KUKA KRL program: EPS_2_25362_MH3A_A_20251103083056.src

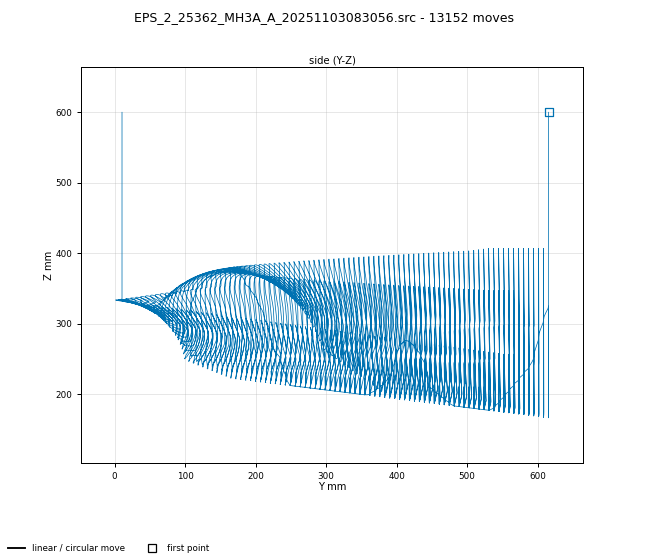
[picture p0: tool path of EPS_2_25362_MH3A_A_20251103083056.src, 13152 of 13154 moves have a stored position in this frame; points joined in program order, loops and branches not executed]
&ACCESS RVP
&REL 4
&COMMENT QRS 19112012
&PARAM EDITMASK = *
DEF PART()
EXT BAS (BAS_COMMAND :IN,REAL :IN )
INT I
BAS (#INITMOV,0 )

;KUKA QRS Post kuka4.cps  Date:22-06-2017 !

File_ID=2900

QRS_PRE_INIT()

;Init var - Until changes are made in qrs_pre_init
Outlet_Square_prg=0
Inlet_1_Square_prg=0
Inlet_2_Square_prg=0
Inlet_3_Square_prg=0
Inlet_4_Square_prg=0
Inlet_5_Square_prg=0

Outlet_1={X 0.000, Y 531.880, Z 306.500, B 0.000, E1 0.000 }
Inlet_1={X 0.000, Y 536.220, Z 246.500, B 0.000, E1 90.000 }
Inlet_2={X 0.000, Y 550.320, Z 206.500, B 0.000, E1 180.000 }
Outlet_1_type=201
Inlet_1_type=201
Inlet_2_type=101
;QRS#1=Sidecore dimensions
;QRS#2=200-8" PVC SDR 35
;QRS#3=200-8" PVC SDR 35
;QRS#4=100-4" PVC SDR 28
;QRS#5=
;QRS#6=
;QRS#7=
;QRS#8=
;QRS#9=12-08 PSX
;QRS#10=12-08 PSX
;QRS#11=8QRS PSX
;QRS#12=
;QRS#13=
;QRS#14=
;QRS#15=
;QRS#16=1220x127x686 2,25'
;QRS#17=EPS Height
;QRS#18=407
;QRS#19=*
;QRS#20= UPDATED VERSION 22-06-2017
;QRS#21=*
Outlet_Square=0100
Inlet_1_Square=0100
Inlet_2_Square=045
Inlet_3_Square=0
Inlet_4_Square=0
Inlet_5_Square=0
Mill_Square=1
Outlet_Square_Prg=204
Inlet_1_Square_prg=204
Inlet_2_Square_prg=201

QRS_INIT()

$ADVANCE=5

; T1
PTP {E1 173.498,E2 173.498}
PTP {X 0,Y 615.498,A -85,B 0,C 180,E1 173.498,E2 173.498,E3 0,E4 0,E5 0,E6 0}
QRS_SPEED_INIT()
LIN {X 0,Y 615.498,Z 600,A -85,B 0,C 180,E1 173.498,E2 173.498,E3 0,E4 0,E5 0,E6 0} C_VEL
LIN {X 0,Y 615.498,Z 337.732,A -85,B 0,C 180,E1 173.498,E2 173.498} C_VEL
LIN {X 0,Y 615.498,Z 326.853,A -85,B 0,C 180,E1 173.498,E2 173.498} C_VEL
LIN {X 0,Y 615.496,Z 325.209,A -85,B 0,C 180,E1 173.418,E2 173.418} C_VEL
LIN {X 0,Y 615.497,Z 317.536,A -85,B 0,C 180,E1 172.455,E2 172.455} C_VEL
LIN {X 0,Y 615.498,Z 307.758,A -85,B 0,C 180,E1 171.463,E2 171.463} C_VEL
LIN {X 0,Y 615.498,Z 297.492,A -85,B 0,C 180,E1 170.636,E2 170.636} C_VEL
LIN {X 0,Y 615.449,Z 285.935,A -85,B 0,C 180,E1 169.888,E2 169.888} C_VEL
LIN {X 0,Y 615.45,Z 274.237,A -85,B 0,C 180,E1 169.299,E2 169.299} C_VEL
LIN {X 0,Y 615.495,Z 262.393,A -85,B 0,C 180,E1 168.847,E2 168.847} C_VEL
LIN {X 0,Y 615.488,Z 250.38,A -85,B 0,C 180,E1 168.515,E2 168.515} C_VEL
LIN {X 0,Y 615.473,Z 240.081,A -85,B 0,C 180,E1 168.306,E2 168.306} C_VEL
LIN {X 0,Y 615.432,Z 231.733,A -85,B 0,C 180,E1 165.768,E2 165.768} C_VEL
LIN {X 0,Y 615.485,Z 222.926,A -85,B 0,C 180,E1 163.072,E2 163.072} C_VEL
LIN {X 0,Y 615.428,Z 214.085,A -85,B 0,C 180,E1 160.313,E2 160.313} C_VEL
LIN {X 0,Y 615.422,Z 206.32,A -85,B 0,C 180,E1 157.861,E2 157.861} C_VEL
LIN {X 0,Y 615.473,Z 197.446,A -85,B 0,C 180,E1 155.007,E2 155.007} C_VEL
LIN {X 0,Y 615.429,Z 189.685,A -85,B 0,C 180,E1 152.451,E2 152.451} C_VEL
LIN {X 0,Y 615.495,Z 181.752,A -85,B 0,C 180,E1 149.84,E2 149.84} C_VEL
LIN {X 0,Y 615.493,Z 173.403,A -85,B 0,C 180,E1 147.154,E2 147.154} C_VEL
LIN {X 0,Y 615.459,Z 166.7,A -85,B 0,C 180,E1 144.983,E2 144.983} C_VEL
LIN {X 0,Y 615.455,Z 166.697,A -85,B 0,C 180,E1 142.755,E2 142.755} C_VEL
LIN {X 0,Y 615.482,Z 166.691,A -85,B 0,C 180,E1 139.912,E2 139.912} C_VEL
LIN {X 0,Y 615.499,Z 166.691,A -85,B 0,C 180,E1 137.648,E2 137.648} C_VEL
LIN {X 0,Y 615.44,Z 166.7,A -85,B 0,C 180,E1 134.927,E2 134.927} C_VEL
LIN {X 0,Y 615.493,Z 166.697,A -85,B 0,C 180,E1 132.353,E2 132.353} C_VEL
LIN {X 0,Y 615.492,Z 166.691,A -85,B 0,C 180,E1 129.75,E2 129.75} C_VEL
LIN {X 0,Y 615.44,Z 166.7,A -85,B 0,C 180,E1 126.93,E2 126.93} C_VEL
LIN {X 0,Y 615.468,Z 166.701,A -85,B 0,C 180,E1 124.697,E2 124.697} C_VEL
LIN {X 0,Y 615.489,Z 166.691,A -85,B 0,C 180,E1 122.33,E2 122.33} C_VEL
LIN {X 0,Y 615.494,Z 166.701,A -85,B 0,C 180,E1 119.795,E2 119.795} C_VEL
LIN {X 0,Y 615.491,Z 170.653,A -85,B 0,C 180,E1 117.045,E2 117.045} C_VEL
LIN {X 0,Y 615.49,Z 174.728,A -85,B 0,C 180,E1 114.273,E2 114.273} C_VEL
LIN {X 0,Y 615.467,Z 179.104,A -85,B 0,C 180,E1 111.433,E2 111.433} C_VEL
LIN {X 0,Y 615.482,Z 183.48,A -85,B 0,C 180,E1 108.647,E2 108.647} C_VEL
LIN {X 0,Y 615.48,Z 187.851,A -85,B 0,C 180,E1 105.906,E2 105.906} C_VEL
LIN {X 0,Y 615.448,Z 192.229,A -85,B 0,C 180,E1 103.203,E2 103.203} C_VEL
LIN {X 0,Y 615.496,Z 196.599,A -85,B 0,C 180,E1 100.528,E2 100.528} C_VEL
LIN {X 0,Y 615.436,Z 200.972,A -85,B 0,C 180,E1 97.877,E2 97.877} C_VEL
LIN {X 0,Y 615.491,Z 202.929,A -85,B 0,C 180,E1 96.693,E2 96.693} C_VEL
LIN {X 0,Y 615.467,Z 211.517,A -85,B 0,C 180,E1 96.393,E2 96.393} C_VEL
LIN {X 0,Y 615.433,Z 219.944,A -85,B 0,C 180,E1 95.982,E2 95.982} C_VEL
LIN {X 0,Y 615.434,Z 227.673,A -85,B 0,C 180,E1 95.489,E2 95.489} C_VEL
LIN {X 0,Y 615.485,Z 234.509,A -85,B 0,C 180,E1 94.914,E2 94.914} C_VEL
LIN {X 0,Y 615.497,Z 240.661,A -85,B 0,C 180,E1 94.257,E2 94.257} C_VEL
LIN {X 0,Y 615.497,Z 245.51,A -85,B 0,C 180,E1 93.601,E2 93.601} C_VEL
LIN {X 0,Y 615.498,Z 249.246,A -85,B 0,C 180,E1 92.946,E2 92.946} C_VEL
LIN {X 0,Y 615.498,Z 253.227,A -85,B 0,C 180,E1 91.964,E2 91.964} C_VEL
LIN {X 0,Y 615.496,Z 254.962,A -85,B 0,C 180,E1 91.309,E2 91.309} C_VEL
LIN {X 0,Y 615.496,Z 256.003,A -85,B 0,C 180,E1 90.655,E2 90.655} C_VEL
LIN {X 0,Y 615.494,Z 256.384,A -85,B 0,C 180,E1 90.001,E2 90.001} C_VEL
LIN {X 0,Y 615.496,Z 256.106,A -85,B 0,C 180,E1 89.347,E2 89.347} C_VEL
LIN {X 0,Y 615.497,Z 255.167,A -85,B 0,C 180,E1 88.692,E2 88.692} C_VEL
LIN {X 0,Y 615.496,Z 253.539,A -85,B 0,C 180,E1 88.038,E2 88.038} C_VEL
LIN {X 0,Y 615.497,Z 251.17,A -85,B 0,C 180,E1 87.383,E2 87.383} C_VEL
LIN {X 0,Y 615.498,Z 246.077,A -85,B 0,C 180,E1 86.4,E2 86.4} C_VEL
LIN {X 0,Y 615.498,Z 240.038,A -85,B 0,C 180,E1 85.58,E2 85.58} C_VEL
LIN {X 0,Y 615.468,Z 233.768,A -85,B 0,C 180,E1 84.924,E2 84.924} C_VEL
LIN {X 0,Y 615.422,Z 226.618,A -85,B 0,C 180,E1 84.348,E2 84.348} C_VEL
LIN {X 0,Y 615.432,Z 218.637,A -85,B 0,C 180,E1 83.855,E2 83.855} C_VEL
LIN {X 0,Y 615.473,Z 209.487,A -85,B 0,C 180,E1 83.437,E2 83.437} C_VEL
LIN {X 0,Y 615.499,Z 202.92,A -85,B 0,C 180,E1 83.213,E2 83.213} C_VEL
LIN {X 0,Y 615.447,Z 198.945,A -85,B 0,C 180,E1 80.802,E2 80.802} C_VEL
LIN {X 0,Y 615.446,Z 195.663,A -85,B 0,C 180,E1 78.807,E2 78.807} C_VEL
LIN {X 0,Y 615.443,Z 192.381,A -85,B 0,C 180,E1 76.799,E2 76.799} C_VEL
LIN {X 0,Y 615.445,Z 189.098,A -85,B 0,C 180,E1 74.774,E2 74.774} C_VEL
LIN {X 0,Y 615.484,Z 184.718,A -85,B 0,C 180,E1 72.044,E2 72.044} C_VEL
LIN {X 0,Y 615.47,Z 180.343,A -85,B 0,C 180,E1 69.27,E2 69.27} C_VEL
LIN {X 0,Y 615.48,Z 175.962,A -85,B 0,C 180,E1 66.445,E2 66.445} C_VEL
LIN {X 0,Y 615.493,Z 171.632,A -85,B 0,C 180,E1 63.557,E2 63.557} C_VEL
LIN {X 0,Y 615.493,Z 168.479,A -85,B 0,C 180,E1 61.344,E2 61.344} C_VEL
LIN {X 0,Y 615.497,Z 166.83,A -85,B 0,C 180,E1 60.204,E2 60.204} C_VEL
LIN {X 0,Y 615.464,Z 166.689,A -85,B 0,C 180,E1 57.543,E2 57.543} C_VEL
LIN {X 0,Y 615.454,Z 166.693,A -85,B 0,C 180,E1 55.184,E2 55.184} C_VEL
LIN {X 0,Y 615.479,Z 166.7,A -85,B 0,C 180,E1 52.759,E2 52.759} C_VEL
LIN {X 0,Y 615.48,Z 166.686,A -85,B 0,C 180,E1 49.912,E2 49.912} C_VEL
LIN {X 0,Y 615.463,Z 166.69,A -85,B 0,C 180,E1 47.647,E2 47.647} C_VEL
LIN {X 0,Y 615.498,Z 166.699,A -85,B 0,C 180,E1 44.934,E2 44.934} C_VEL
LIN {X 0,Y 615.475,Z 166.686,A -85,B 0,C 180,E1 42.081,E2 42.081} C_VEL
LIN {X 0,Y 615.47,Z 166.692,A -85,B 0,C 180,E1 39.752,E2 39.752} C_VEL
LIN {X 0,Y 615.484,Z 166.691,A -85,B 0,C 180,E1 36.938,E2 36.938} C_VEL
LIN {X 0,Y 615.489,Z 166.684,A -85,B 0,C 180,E1 34.703,E2 34.703} C_VEL
LIN {X 0,Y 615.481,Z 166.686,A -85,B 0,C 180,E1 32.332,E2 32.332} C_VEL
LIN {X 0,Y 615.489,Z 166.698,A -85,B 0,C 180,E1 29.797,E2 29.797} C_VEL
LIN {X 0,Y 615.477,Z 166.687,A -85,B 0,C 180,E1 27.046,E2 27.046} C_VEL
LIN {X 0,Y 615.483,Z 166.693,A -85,B 0,C 180,E1 24.272,E2 24.272} C_VEL
LIN {X 0,Y 615.472,Z 166.69,A -85,B 0,C 180,E1 21.433,E2 21.433} C_VEL
LIN {X 0,Y 615.486,Z 166.69,A -85,B 0,C 180,E1 18.608,E2 18.608} C_VEL
LIN {X 0,Y 615.471,Z 166.694,A -85,B 0,C 180,E1 15.906,E2 15.906} C_VEL
LIN {X 0,Y 615.49,Z 166.684,A -85,B 0,C 180,E1 13.201,E2 13.201} C_VEL
LIN {X 0,Y 615.489,Z 166.702,A -85,B 0,C 180,E1 10.527,E2 10.527} C_VEL
LIN {X 0,Y 615.459,Z 166.691,A -85,B 0,C 180,E1 7.876,E2 7.876} C_VEL
LIN {X 0,Y 615.496,Z 166.688,A -85,B 0,C 180,E1 5.241,E2 5.241} C_VEL
LIN {X 0,Y 615.47,Z 166.697,A -85,B 0,C 180,E1 2.618,E2 2.618} C_VEL
LIN {X 0,Y 615.456,Z 166.691,A -85,B 0,C 180,E1 0,E2 0} C_VEL
LIN {X 0,Y 615.495,Z 166.693,A -85,B 0,C 180,E1 -2.618,E2 -2.618} C_VEL
LIN {X 0,Y 615.451,Z 166.697,A -85,B 0,C 180,E1 -5.242,E2 -5.242} C_VEL
LIN {X 0,Y 615.446,Z 166.696,A -85,B 0,C 180,E1 -7.216,E2 -7.216} C_VEL
LIN {X 0,Y 615.442,Z 166.696,A -85,B 0,C 180,E1 -9.199,E2 -9.199} C_VEL
LIN {X 0,Y 615.437,Z 166.696,A -85,B 0,C 180,E1 -11.194,E2 -11.194} C_VEL
LIN {X 0,Y 615.473,Z 166.694,A -85,B 0,C 180,E1 -13.933,E2 -13.933} C_VEL
LIN {X 0,Y 615.453,Z 166.699,A -85,B 0,C 180,E1 -16.588,E2 -16.588} C_VEL
LIN {X 0,Y 615.439,Z 166.699,A -85,B 0,C 180,E1 -18.648,E2 -18.648} C_VEL
LIN {X 0,Y 615.427,Z 166.699,A -85,B 0,C 180,E1 -20.733,E2 -20.733} C_VEL
LIN {X 0,Y 615.419,Z 166.699,A -85,B 0,C 180,E1 -22.847,E2 -22.847} C_VEL
LIN {X 0,Y 615.418,Z 166.7,A -85,B 0,C 180,E1 -24.995,E2 -24.995} C_VEL
LIN {X 0,Y 615.433,Z 166.7,A -85,B 0,C 180,E1 -27.18,E2 -27.18} C_VEL
LIN {X 0,Y 615.438,Z 166.698,A -85,B 0,C 180,E1 -30.163,E2 -30.163} C_VEL
LIN {X 0,Y 615.424,Z 166.698,A -85,B 0,C 180,E1 -32.461,E2 -32.461} C_VEL
LIN {X 0,Y 615.438,Z 166.699,A -85,B 0,C 180,E1 -34.818,E2 -34.818} C_VEL
LIN {X 0,Y 615.488,Z 166.702,A -85,B 0,C 180,E1 -37.242,E2 -37.242} C_VEL
LIN {X 0,Y 615.457,Z 166.694,A -85,B 0,C 180,E1 -39.753,E2 -39.753} C_VEL
LIN {X 0,Y 615.44,Z 166.696,A -85,B 0,C 180,E1 -42.357,E2 -42.357} C_VEL
LIN {X 0,Y 615.491,Z 166.696,A -85,B 0,C 180,E1 -45.068,E2 -45.068} C_VEL
LIN {X 0,Y 615.454,Z 166.692,A -85,B 0,C 180,E1 -47.646,E2 -47.646} C_VEL
LIN {X 0,Y 615.456,Z 166.697,A -85,B 0,C 180,E1 -50.249,E2 -50.249} C_VEL
LIN {X 0,Y 615.487,Z 166.688,A -85,B 0,C 180,E1 -53.064,E2 -53.064} C_VEL
LIN {X 0,Y 615.467,Z 166.689,A -85,B 0,C 180,E1 -55.303,E2 -55.303} C_VEL
LIN {X 0,Y 615.456,Z 166.693,A -85,B 0,C 180,E1 -57.674,E2 -57.674} C_VEL
LIN {X 0,Y 615.497,Z 166.7,A -85,B 0,C 180,E1 -60.204,E2 -60.204} C_VEL
LIN {X 0,Y 615.46,Z 166.871,A -85,B 0,C 180,E1 -61.448,E2 -61.448} C_VEL
LIN {X 0,Y 615.473,Z 186.055,A -85,B 0,C 180,E1 -64.103,E2 -64.103} C_VEL
LIN {X 0,Y 615.484,Z 205.999,A -85,B 0,C 180,E1 -66.801,E2 -66.801} C_VEL
LIN {X 0,Y 615.469,Z 225.967,A -85,B 0,C 180,E1 -69.448,E2 -69.448} C_VEL
LIN {X 0,Y 615.482,Z 247.188,A -85,B 0,C 180,E1 -72.216,E2 -72.216} C_VEL
LIN {X 0,Y 615.481,Z 268.409,A -85,B 0,C 180,E1 -74.944,E2 -74.944} C_VEL
LIN {X 0,Y 615.47,Z 289.61,A -85,B 0,C 180,E1 -77.638,E2 -77.638} C_VEL
LIN {X 0,Y 615.498,Z 294.736,A -85,B 0,C 180,E1 -78.287,E2 -78.287} C_VEL
LIN {X 0,Y 615.483,Z 310.284,A -85,B 0,C 180,E1 -78.558,E2 -78.558} C_VEL
LIN {X 0,Y 615.479,Z 323.353,A -85,B 0,C 180,E1 -78.922,E2 -78.922} C_VEL
LIN {X 0,Y 615.487,Z 335.144,A -85,B 0,C 180,E1 -79.384,E2 -79.384} C_VEL
LIN {X 0,Y 615.481,Z 346.592,A -85,B 0,C 180,E1 -79.973,E2 -79.973} C_VEL
LIN {X 0,Y 615.499,Z 358.034,A -85,B 0,C 180,E1 -80.719,E2 -80.719} C_VEL
LIN {X 0,Y 615.498,Z 367.268,A -85,B 0,C 180,E1 -81.464,E2 -81.464} C_VEL
LIN {X 0,Y 615.5,Z 375.662,A -85,B 0,C 180,E1 -82.291,E2 -82.291} C_VEL
LIN {X 0,Y 615.497,Z 383.692,A -85,B 0,C 180,E1 -83.259,E2 -83.259} C_VEL
LIN {X 0,Y 615.499,Z 389.428,A -85,B 0,C 180,E1 -84.102,E2 -84.102} C_VEL
LIN {X 0,Y 615.496,Z 394.877,A -85,B 0,C 180,E1 -85.088,E2 -85.088} C_VEL
LIN {X 0,Y 615.497,Z 399.144,A -85,B 0,C 180,E1 -86.072,E2 -86.072} C_VEL
LIN {X 0,Y 615.494,Z 401.401,A -85,B 0,C 180,E1 -86.728,E2 -86.728} C_VEL
LIN {X 0,Y 615.497,Z 403.235,A -85,B 0,C 180,E1 -87.383,E2 -87.383} C_VEL
LIN {X 0,Y 615.5,Z 404.609,A -85,B 0,C 180,E1 -88.038,E2 -88.038} C_VEL
LIN {X 0,Y 615.496,Z 406.174,A -85,B 0,C 180,E1 -89.347,E2 -89.347} C_VEL
LIN {X 0,Y 615.494,Z 406.389,A -85,B 0,C 180,E1 -90.001,E2 -90.001} C_VEL
LIN {X 0,Y 615.495,Z 405.579,A -85,B 0,C 180,E1 -91.309,E2 -91.309} C_VEL
LIN {X 0,Y 615.5,Z 404.606,A -85,B 0,C 180,E1 -91.964,E2 -91.964} C_VEL
LIN {X 0,Y 615.497,Z 403.231,A -85,B 0,C 180,E1 -92.619,E2 -92.619} C_VEL
LIN {X 0,Y 615.496,Z 400.347,A -85,B 0,C 180,E1 -93.601,E2 -93.601} C_VEL
LIN {X 0,Y 615.498,Z 396.438,A -85,B 0,C 180,E1 -94.585,E2 -94.585} C_VEL
LIN {X 0,Y 615.499,Z 391.4,A -85,B 0,C 180,E1 -95.57,E2 -95.57} C_VEL
LIN {X 0,Y 615.497,Z 384.87,A -85,B 0,C 180,E1 -96.583,E2 -96.583} C_VEL
LIN {X 0,Y 615.497,Z 377.126,A -85,B 0,C 180,E1 -97.546,E2 -97.546} C_VEL
LIN {X 0,Y 615.498,Z 369.037,A -85,B 0,C 180,E1 -98.372,E2 -98.372} C_VEL
LIN {X 0,Y 615.499,Z 359.157,A -85,B 0,C 180,E1 -99.199,E2 -99.199} C_VEL
LIN {X 0,Y 615.485,Z 347.969,A -85,B 0,C 180,E1 -99.946,E2 -99.946} C_VEL
LIN {X 0,Y 615.485,Z 337.007,A -85,B 0,C 180,E1 -100.528,E2 -100.528} C_VEL
LIN {X 0,Y 615.479,Z 324.491,A -85,B 0,C 180,E1 -101.04,E2 -101.04} C_VEL
LIN {X 0,Y 615.481,Z 312.033,A -85,B 0,C 180,E1 -101.402,E2 -101.402} C_VEL
LIN {X 0,Y 615.497,Z 298.409,A -85,B 0,C 180,E1 -101.653,E2 -101.653} C_VEL
LIN {X 0,Y 615.498,Z 294.722,A -85,B 0,C 180,E1 -101.715,E2 -101.715} C_VEL
LIN {X 0,Y 615.472,Z 272.374,A -85,B 0,C 180,E1 -104.55,E2 -104.55} C_VEL
LIN {X 0,Y 615.481,Z 251.154,A -85,B 0,C 180,E1 -107.271,E2 -107.271} C_VEL
LIN {X 0,Y 615.481,Z 229.912,A -85,B 0,C 180,E1 -110.034,E2 -110.034} C_VEL
LIN {X 0,Y 615.471,Z 210.527,A -85,B 0,C 180,E1 -112.595,E2 -112.595} C_VEL
LIN {X 0,Y 615.498,Z 189.5,A -85,B 0,C 180,E1 -115.425,E2 -115.425} C_VEL
LIN {X 0,Y 615.471,Z 169.523,A -85,B 0,C 180,E1 -118.18,E2 -118.18} C_VEL
LIN {X 0,Y 615.46,Z 166.693,A -85,B 0,C 180,E1 -118.606,E2 -118.606} C_VEL
LIN {X 0,Y 615.484,Z 166.694,A -85,B 0,C 180,E1 -121.085,E2 -121.085} C_VEL
LIN {X 0,Y 615.427,Z 166.7,A -85,B 0,C 180,E1 -124.026,E2 -124.026} C_VEL
LIN {X 0,Y 615.488,Z 166.696,A -85,B 0,C 180,E1 -126.936,E2 -126.936} C_VEL
LIN {X 0,Y 615.459,Z 166.695,A -85,B 0,C 180,E1 -129.753,E2 -129.753} C_VEL
LIN {X 0,Y 615.488,Z 166.694,A -85,B 0,C 180,E1 -132.354,E2 -132.354} C_VEL
LIN {X 0,Y 615.484,Z 166.69,A -85,B 0,C 180,E1 -135.069,E2 -135.069} C_VEL
LIN {X 0,Y 615.476,Z 166.697,A -85,B 0,C 180,E1 -137.646,E2 -137.646} C_VEL
LIN {X 0,Y 615.465,Z 166.692,A -85,B 0,C 180,E1 -140.248,E2 -140.248} C_VEL
LIN {X 0,Y 615.452,Z 166.7,A -85,B 0,C 180,E1 -143.068,E2 -143.068} C_VEL
LIN {X 0,Y 615.433,Z 166.7,A -85,B 0,C 180,E1 -145.642,E2 -145.642} C_VEL
LIN {X 0,Y 615.449,Z 166.873,A -85,B 0,C 180,E1 -145.893,E2 -145.893} C_VEL
LIN {X 0,Y 615.494,Z 175.891,A -85,B 0,C 180,E1 -148.315,E2 -148.315} C_VEL
LIN {X 0,Y 615.464,Z 184.98,A -85,B 0,C 180,E1 -150.967,E2 -150.967} C_VEL
LIN {X 0,Y 615.489,Z 192.732,A -85,B 0,C 180,E1 -153.556,E2 -153.556} C_VEL
LIN {X 0,Y 615.479,Z 201.605,A -85,B 0,C 180,E1 -156.443,E2 -156.443} C_VEL
LIN {X 0,Y 615.491,Z 210.458,A -85,B 0,C 180,E1 -159.269,E2 -159.269} C_VEL
LIN {X 0,Y 615.492,Z 219.321,A -85,B 0,C 180,E1 -162.043,E2 -162.043} C_VEL
LIN {X 0,Y 615.49,Z 228.167,A -85,B 0,C 180,E1 -164.774,E2 -164.774} C_VEL
LIN {X 0,Y 615.474,Z 237.019,A -85,B 0,C 180,E1 -167.47,E2 -167.47} C_VEL
LIN {X 0,Y 615.487,Z 240.126,A -85,B 0,C 180,E1 -168.411,E2 -168.411} C_VEL
LIN {X 0,Y 615.492,Z 253.696,A -85,B 0,C 180,E1 -168.682,E2 -168.682} C_VEL
LIN {X 0,Y 615.468,Z 266.631,A -85,B 0,C 180,E1 -169.084,E2 -169.084} C_VEL
LIN {X 0,Y 615.479,Z 277.823,A -85,B 0,C 180,E1 -169.556,E2 -169.556} C_VEL
LIN {X 0,Y 615.489,Z 290.02,A -85,B 0,C 180,E1 -170.221,E2 -170.221} C_VEL
LIN {X 0,Y 615.498,Z 300.713,A -85,B 0,C 180,E1 -170.967,E2 -170.967} C_VEL
LIN {X 0,Y 615.498,Z 310.33,A -85,B 0,C 180,E1 -171.794,E2 -171.794} C_VEL
LIN {X 0,Y 615.497,Z 318.209,A -85,B 0,C 180,E1 -172.62,E2 -172.62} C_VEL
LIN {X 0,Y 615.497,Z 325.899,A -85,B 0,C 180,E1 -173.608,E2 -173.608} C_VEL
LIN {X 0,Y 615.497,Z 332.958,A -85,B 0,C 180,E1 -174.759,E2 -174.759} C_VEL
LIN {X 0,Y 615.498,Z 337.657,A -85,B 0,C 180,E1 -175.744,E2 -175.744} C_VEL
LIN {X 0,Y 615.494,Z 341.255,A -85,B 0,C 180,E1 -176.727,E2 -176.727} C_VEL
LIN {X 0,Y 615.496,Z 343.115,A -85,B 0,C 180,E1 -177.382,E2 -177.382} C_VEL
LIN {X 0,Y 615.497,Z 344.533,A -85,B 0,C 180,E1 -178.037,E2 -178.037} C_VEL
LIN {X 0,Y 615.497,Z 346.141,A -85,B 0,C 180,E1 -179.346,E2 -179.346} C_VEL
LIN {X 0,Y 615.494,Z 346.384,A -85,B 0,C 180,E1 -180,E2 -180} C_VEL
LIN {X 0,Y 615.495,Z 346.206,A -85,B 0,C 180,E1 -180.654,E2 -180.654} C_VEL
LIN {X 0,Y 615.496,Z 344.683,A -85,B 0,C 180,E1 -181.963,E2 -181.963} C_VEL
LIN {X 0,Y 615.498,Z 343.341,A -85,B 0,C 180,E1 -182.618,E2 -182.618} C_VEL
LIN {X 0,Y 615.497,Z 340.494,A -85,B 0,C 180,E1 -183.601,E2 -183.601} C_VEL
LIN {X 0,Y 615.498,Z 336.634,A -85,B 0,C 180,E1 -184.585,E2 -184.585} C_VEL
LIN {X 0,Y 615.498,Z 331.651,A -85,B 0,C 180,E1 -185.57,E2 -185.57} C_VEL
LIN {X 0,Y 615.496,Z 325.209,A -85,B 0,C 180,E1 -186.582,E2 -186.582} C_VEL
LIN {X 0,Y 614.829,Z 322.027,A -85,B 0,C 180,E1 -187.031,E2 -187.031} C_VEL
LIN {X 0,Y 611.989,Z 316.454,A -85,B 0,C 180,E1 -187.748,E2 -187.748} C_VEL
LIN {X 0,Y 609.138,Z 310.179,A -85,B 0,C 180,E1 -188.429,E2 -188.429} C_VEL
LIN {X 0,Y 608.477,Z 305.938,A -85,B 0,C 180,E1 -188.819,E2 -188.819} C_VEL
LIN {X 0,Y 608.49,Z 295.389,A -85,B 0,C 180,E1 -189.641,E2 -189.641} C_VEL
LIN {X 0,Y 608.446,Z 284.609,A -85,B 0,C 180,E1 -190.314,E2 -190.314} C_VEL
LIN {X 0,Y 608.493,Z 272.214,A -85,B 0,C 180,E1 -190.917,E2 -190.917} C_VEL
LIN {X 0,Y 608.556,Z 259.968,A -85,B 0,C 180,E1 -191.365,E2 -191.365} C_VEL
LIN {X 0,Y 608.538,Z 247.651,A -85,B 0,C 180,E1 -191.681,E2 -191.681} C_VEL
LIN {X 0,Y 608.425,Z 240.5,A -85,B 0,C 180,E1 -191.81,E2 -191.81} C_VEL
LIN {X 0,Y 608.384,Z 232.081,A -85,B 0,C 180,E1 -194.381,E2 -194.381} C_VEL
LIN {X 0,Y 608.444,Z 223.175,A -85,B 0,C 180,E1 -197.13,E2 -197.13} C_VEL
LIN {X 0,Y 608.394,Z 214.268,A -85,B 0,C 180,E1 -199.924,E2 -199.924} C_VEL
LIN {X 0,Y 608.433,Z 206.281,A -85,B 0,C 180,E1 -202.469,E2 -202.469} C_VEL
LIN {X 0,Y 608.417,Z 197.567,A -85,B 0,C 180,E1 -205.303,E2 -205.303} C_VEL
LIN {X 0,Y 608.417,Z 189.772,A -85,B 0,C 180,E1 -207.894,E2 -207.894} C_VEL
LIN {X 0,Y 608.488,Z 181.66,A -85,B 0,C 180,E1 -210.544,E2 -210.544} C_VEL
LIN {X 0,Y 608.475,Z 173.202,A -85,B 0,C 180,E1 -213.274,E2 -213.274} C_VEL
LIN {X 0,Y 608.433,Z 167.696,A -85,B 0,C 180,E1 -215.062,E2 -215.062} C_VEL
LIN {X 0,Y 608.463,Z 167.695,A -85,B 0,C 180,E1 -217.747,E2 -217.747} C_VEL
LIN {X 0,Y 608.451,Z 167.691,A -85,B 0,C 180,E1 -220.328,E2 -220.328} C_VEL
LIN {X 0,Y 608.432,Z 167.697,A -85,B 0,C 180,E1 -222.962,E2 -222.962} C_VEL
LIN {X 0,Y 608.456,Z 167.695,A -85,B 0,C 180,E1 -225.736,E2 -225.736} C_VEL
LIN {X 0,Y 608.459,Z 167.692,A -85,B 0,C 180,E1 -228.658,E2 -228.658} C_VEL
LIN {X 0,Y 608.461,Z 167.691,A -85,B 0,C 180,E1 -231.761,E2 -231.761} C_VEL
LIN {X 0,Y 608.419,Z 167.695,A -85,B 0,C 180,E1 -234.72,E2 -234.72} C_VEL
LIN {X 0,Y 608.463,Z 167.692,A -85,B 0,C 180,E1 -237.478,E2 -237.478} C_VEL
LIN {X 0,Y 608.478,Z 167.693,A -85,B 0,C 180,E1 -240.22,E2 -240.22} C_VEL
LIN {X 0,Y 608.433,Z 171.873,A -85,B 0,C 180,E1 -243.224,E2 -243.224} C_VEL
LIN {X 0,Y 608.43,Z 175.706,A -85,B 0,C 180,E1 -245.858,E2 -245.858} C_VEL
LIN {X 0,Y 608.404,Z 179.457,A -85,B 0,C 180,E1 -248.305,E2 -248.305} C_VEL
LIN {X 0,Y 608.399,Z 182.761,A -85,B 0,C 180,E1 -250.427,E2 -250.427} C_VEL
LIN {X 0,Y 608.394,Z 186.065,A -85,B 0,C 180,E1 -252.521,E2 -252.521} C_VEL
LIN {X 0,Y 608.408,Z 190.471,A -85,B 0,C 180,E1 -255.277,E2 -255.277} C_VEL
LIN {X 0,Y 608.411,Z 194.877,A -85,B 0,C 180,E1 -257.998,E2 -257.998} C_VEL
LIN {X 0,Y 608.392,Z 198.181,A -85,B 0,C 180,E1 -260.021,E2 -260.021} C_VEL
LIN {X 0,Y 608.384,Z 202.587,A -85,B 0,C 180,E1 -262.699,E2 -262.699} C_VEL
LIN {X 0,Y 608.442,Z 203.457,A -85,B 0,C 180,E1 -263.226,E2 -263.226} C_VEL
LIN {X 0,Y 608.431,Z 212.066,A -85,B 0,C 180,E1 -263.533,E2 -263.533} C_VEL
LIN {X 0,Y 608.391,Z 220.456,A -85,B 0,C 180,E1 -263.948,E2 -263.948} C_VEL
LIN {X 0,Y 608.403,Z 228.169,A -85,B 0,C 180,E1 -264.447,E2 -264.447} C_VEL
LIN {X 0,Y 608.457,Z 235.022,A -85,B 0,C 180,E1 -265.029,E2 -265.029} C_VEL
LIN {X 0,Y 608.443,Z 241.199,A -85,B 0,C 180,E1 -265.693,E2 -265.693} C_VEL
LIN {X 0,Y 608.451,Z 246.062,A -85,B 0,C 180,E1 -266.357,E2 -266.357} C_VEL
LIN {X 0,Y 608.452,Z 249.816,A -85,B 0,C 180,E1 -267.02,E2 -267.02} C_VEL
LIN {X 0,Y 608.443,Z 253.823,A -85,B 0,C 180,E1 -268.013,E2 -268.013} C_VEL
LIN {X 0,Y 608.448,Z 255.566,A -85,B 0,C 180,E1 -268.675,E2 -268.675} C_VEL
LIN {X 0,Y 608.439,Z 256.612,A -85,B 0,C 180,E1 -269.337,E2 -269.337} C_VEL
LIN {X 0,Y 608.434,Z 256.994,A -85,B 0,C 180,E1 -269.999,E2 -269.999} C_VEL
LIN {X 0,Y 608.438,Z 256.715,A -85,B 0,C 180,E1 -270.661,E2 -270.661} C_VEL
LIN {X 0,Y 608.449,Z 255.77,A -85,B 0,C 180,E1 -271.323,E2 -271.323} C_VEL
LIN {X 0,Y 608.442,Z 254.132,A -85,B 0,C 180,E1 -271.985,E2 -271.985} C_VEL
LIN {X 0,Y 608.429,Z 251.75,A -85,B 0,C 180,E1 -272.647,E2 -272.647} C_VEL
LIN {X 0,Y 608.452,Z 246.624,A -85,B 0,C 180,E1 -273.641,E2 -273.641} C_VEL
LIN {X 0,Y 608.451,Z 240.563,A -85,B 0,C 180,E1 -274.471,E2 -274.471} C_VEL
LIN {X 0,Y 608.429,Z 234.262,A -85,B 0,C 180,E1 -275.135,E2 -275.135} C_VEL
LIN {X 0,Y 608.401,Z 227.107,A -85,B 0,C 180,E1 -275.717,E2 -275.717} C_VEL
LIN {X 0,Y 608.39,Z 219.121,A -85,B 0,C 180,E1 -276.216,E2 -276.216} C_VEL
LIN {X 0,Y 608.439,Z 210.281,A -85,B 0,C 180,E1 -276.632,E2 -276.632} C_VEL
LIN {X 0,Y 608.431,Z 203.443,A -85,B 0,C 180,E1 -276.872,E2 -276.872} C_VEL
LIN {X 0,Y 608.371,Z 199.433,A -85,B 0,C 180,E1 -279.306,E2 -279.306} C_VEL
LIN {X 0,Y 608.387,Z 196.128,A -85,B 0,C 180,E1 -281.324,E2 -281.324} C_VEL
LIN {X 0,Y 608.415,Z 191.72,A -85,B 0,C 180,E1 -284.038,E2 -284.038} C_VEL
LIN {X 0,Y 608.406,Z 187.313,A -85,B 0,C 180,E1 -286.784,E2 -286.784} C_VEL
LIN {X 0,Y 608.401,Z 184.007,A -85,B 0,C 180,E1 -288.87,E2 -288.87} C_VEL
LIN {X 0,Y 608.397,Z 180.701,A -85,B 0,C 180,E1 -290.983,E2 -290.983} C_VEL
LIN {X 0,Y 608.401,Z 177.396,A -85,B 0,C 180,E1 -293.125,E2 -293.125} C_VEL
LIN {X 0,Y 608.449,Z 173.08,A -85,B 0,C 180,E1 -296.034,E2 -296.034} C_VEL
LIN {X 0,Y 608.447,Z 169.414,A -85,B 0,C 180,E1 -298.615,E2 -298.615} C_VEL
LIN {X 0,Y 608.461,Z 167.693,A -85,B 0,C 180,E1 -299.97,E2 -299.97} C_VEL
LIN {X 0,Y 608.44,Z 167.69,A -85,B 0,C 180,E1 -302.879,E2 -302.879} C_VEL
LIN {X 0,Y 608.436,Z 167.697,A -85,B 0,C 180,E1 -305.277,E2 -305.277} C_VEL
LIN {X 0,Y 608.465,Z 167.691,A -85,B 0,C 180,E1 -307.745,E2 -307.745} C_VEL
LIN {X 0,Y 608.436,Z 167.69,A -85,B 0,C 180,E1 -310.327,E2 -310.327} C_VEL
LIN {X 0,Y 608.48,Z 167.691,A -85,B 0,C 180,E1 -313.309,E2 -313.309} C_VEL
LIN {X 0,Y 608.462,Z 167.687,A -85,B 0,C 180,E1 -316.13,E2 -316.13} C_VEL
LIN {X 0,Y 608.453,Z 167.698,A -85,B 0,C 180,E1 -318.823,E2 -318.823} C_VEL
LIN {X 0,Y 608.464,Z 167.688,A -85,B 0,C 180,E1 -321.411,E2 -321.411} C_VEL
LIN {X 0,Y 608.468,Z 167.687,A -85,B 0,C 180,E1 -323.95,E2 -323.95} C_VEL
LIN {X 0,Y 608.466,Z 167.693,A -85,B 0,C 180,E1 -326.329,E2 -326.329} C_VEL
LIN {X 0,Y 608.47,Z 167.691,A -85,B 0,C 180,E1 -328.726,E2 -328.726} C_VEL
LIN {X 0,Y 608.472,Z 167.686,A -85,B 0,C 180,E1 -331.378,E2 -331.378} C_VEL
LIN {X 0,Y 608.469,Z 167.694,A -85,B 0,C 180,E1 -334.276,E2 -334.276} C_VEL
LIN {X 0,Y 608.446,Z 167.689,A -85,B 0,C 180,E1 -336.876,E2 -336.876} C_VEL
LIN {X 0,Y 608.463,Z 167.694,A -85,B 0,C 180,E1 -339.726,E2 -339.726} C_VEL
LIN {X 0,Y 608.441,Z 167.69,A -85,B 0,C 180,E1 -342.523,E2 -342.523} C_VEL
LIN {X 0,Y 608.476,Z 167.689,A -85,B 0,C 180,E1 -345.279,E2 -345.279} C_VEL
LIN {X 0,Y 608.444,Z 167.692,A -85,B 0,C 180,E1 -348,E2 -348} C_VEL
LIN {X 0,Y 608.474,Z 167.686,A -85,B 0,C 180,E1 -350.694,E2 -350.694} C_VEL
LIN {X 0,Y 608.465,Z 167.695,A -85,B 0,C 180,E1 -353.367,E2 -353.367} C_VEL
LIN {X 0,Y 608.428,Z 167.691,A -85,B 0,C 180,E1 -356.026,E2 -356.026} C_VEL
LIN {X 0,Y 608.476,Z 167.689,A -85,B 0,C 180,E1 -358.676,E2 -358.676} C_VEL
LIN {X 0,Y 608.445,Z 167.692,A -85,B 0,C 180,E1 -361.324,E2 -361.324} C_VEL
LIN {X 0,Y 608.45,Z 167.691,A -85,B 0,C 180,E1 -363.311,E2 -363.311} C_VEL
LIN {X 0,Y 608.434,Z 167.691,A -85,B 0,C 180,E1 -365.967,E2 -365.967} C_VEL
LIN {X 0,Y 608.454,Z 167.697,A -85,B 0,C 180,E1 -368.636,E2 -368.636} C_VEL
LIN {X 0,Y 608.412,Z 167.693,A -85,B 0,C 180,E1 -371.325,E2 -371.325} C_VEL
LIN {X 0,Y 608.456,Z 167.693,A -85,B 0,C 180,E1 -374.038,E2 -374.038} C_VEL
LIN {X 0,Y 608.413,Z 167.695,A -85,B 0,C 180,E1 -376.785,E2 -376.785} C_VEL
LIN {X 0,Y 608.419,Z 167.695,A -85,B 0,C 180,E1 -379.572,E2 -379.572} C_VEL
LIN {X 0,Y 608.416,Z 167.695,A -85,B 0,C 180,E1 -382.47,E2 -382.47} C_VEL
LIN {X 0,Y 608.407,Z 167.694,A -85,B 0,C 180,E1 -384.573,E2 -384.573} C_VEL
LIN {X 0,Y 608.386,Z 167.696,A -85,B 0,C 180,E1 -386.777,E2 -386.777} C_VEL
LIN {X 0,Y 608.462,Z 167.694,A -85,B 0,C 180,E1 -389.78,E2 -389.78} C_VEL
LIN {X 0,Y 608.408,Z 167.694,A -85,B 0,C 180,E1 -392.517,E2 -392.517} C_VEL
LIN {X 0,Y 608.409,Z 167.696,A -85,B 0,C 180,E1 -394.902,E2 -394.902} C_VEL
LIN {X 0,Y 608.441,Z 167.692,A -85,B 0,C 180,E1 -397.748,E2 -397.748} C_VEL
LIN {X 0,Y 608.423,Z 167.692,A -85,B 0,C 180,E1 -400.328,E2 -400.328} C_VEL
LIN {X 0,Y 608.451,Z 167.698,A -85,B 0,C 180,E1 -402.96,E2 -402.96} C_VEL
LIN {X 0,Y 608.422,Z 167.692,A -85,B 0,C 180,E1 -405.74,E2 -405.74} C_VEL
LIN {X 0,Y 608.427,Z 167.691,A -85,B 0,C 180,E1 -407.937,E2 -407.937} C_VEL
LIN {X 0,Y 608.472,Z 167.695,A -85,B 0,C 180,E1 -410.703,E2 -410.703} C_VEL
LIN {X 0,Y 608.456,Z 167.69,A -85,B 0,C 180,E1 -413.087,E2 -413.087} C_VEL
LIN {X 0,Y 608.451,Z 167.688,A -85,B 0,C 180,E1 -415.531,E2 -415.531} C_VEL
LIN {X 0,Y 608.449,Z 167.692,A -85,B 0,C 180,E1 -417.906,E2 -417.906} C_VEL
LIN {X 0,Y 608.481,Z 167.695,A -85,B 0,C 180,E1 -420.222,E2 -420.222} C_VEL
LIN {X 0,Y 608.464,Z 167.784,A -85,B 0,C 180,E1 -421.219,E2 -421.219} C_VEL
LIN {X 0,Y 608.697,Z 175.418,A -85,B 0,C 180,E1 -422.309,E2 -422.309} C_VEL
LIN {X 0,Y 608.625,Z 196.691,A -85,B 0,C 180,E1 -425.256,E2 -425.256} C_VEL
LIN {X 0,Y 608.596,Z 216.635,A -85,B 0,C 180,E1 -427.958,E2 -427.958} C_VEL
LIN {X 0,Y 608.553,Z 237.909,A -85,B 0,C 180,E1 -430.785,E2 -430.785} C_VEL
LIN {X 0,Y 608.51,Z 259.293,A -85,B 0,C 180,E1 -433.578,E2 -433.578} C_VEL
LIN {X 0,Y 608.494,Z 281.786,A -85,B 0,C 180,E1 -436.475,E2 -436.475} C_VEL
LIN {X 0,Y 608.493,Z 294.915,A -85,B 0,C 180,E1 -438.15,E2 -438.15} C_VEL
LIN {X 0,Y 608.545,Z 311.309,A -85,B 0,C 180,E1 -438.446,E2 -438.446} C_VEL
LIN {X 0,Y 608.521,Z 323.925,A -85,B 0,C 180,E1 -438.809,E2 -438.809} C_VEL
LIN {X 0,Y 608.515,Z 335.613,A -85,B 0,C 180,E1 -439.276,E2 -439.276} C_VEL
LIN {X 0,Y 608.489,Z 346.772,A -85,B 0,C 180,E1 -439.856,E2 -439.856} C_VEL
LIN {X 0,Y 608.503,Z 358.265,A -85,B 0,C 180,E1 -440.612,E2 -440.612} C_VEL
LIN {X 0,Y 608.472,Z 367.547,A -85,B 0,C 180,E1 -441.365,E2 -441.365} C_VEL
LIN {X 0,Y 608.456,Z 375.997,A -85,B 0,C 180,E1 -442.201,E2 -442.201} C_VEL
LIN {X 0,Y 608.461,Z 384.242,A -85,B 0,C 180,E1 -443.202,E2 -443.202} C_VEL
LIN {X 0,Y 608.438,Z 390.882,A -85,B 0,C 180,E1 -444.2,E2 -444.2} C_VEL
LIN {X 0,Y 608.432,Z 396.954,A -85,B 0,C 180,E1 -445.363,E2 -445.363} C_VEL
LIN {X 0,Y 608.449,Z 400.899,A -85,B 0,C 180,E1 -446.359,E2 -446.359} C_VEL
LIN {X 0,Y 608.425,Z 403.811,A -85,B 0,C 180,E1 -447.353,E2 -447.353} C_VEL
LIN {X 0,Y 608.444,Z 405.203,A -85,B 0,C 180,E1 -448.015,E2 -448.015} C_VEL
LIN {X 0,Y 608.438,Z 406.784,A -85,B 0,C 180,E1 -449.339,E2 -449.339} C_VEL
LIN {X 0,Y 608.434,Z 407,A -85,B 0,C 180,E1 -450.001,E2 -450.001} C_VEL
LIN {X 0,Y 608.448,Z 406.183,A -85,B 0,C 180,E1 -451.325,E2 -451.325} C_VEL
LIN {X 0,Y 608.445,Z 405.2,A -85,B 0,C 180,E1 -451.987,E2 -451.987} C_VEL
LIN {X 0,Y 608.425,Z 403.807,A -85,B 0,C 180,E1 -452.649,E2 -452.649} C_VEL
LIN {X 0,Y 608.449,Z 400.893,A -85,B 0,C 180,E1 -453.643,E2 -453.643} C_VEL
LIN {X 0,Y 608.432,Z 396.947,A -85,B 0,C 180,E1 -454.639,E2 -454.639} C_VEL
LIN {X 0,Y 608.438,Z 390.872,A -85,B 0,C 180,E1 -455.802,E2 -455.802} C_VEL
LIN {X 0,Y 608.463,Z 384.229,A -85,B 0,C 180,E1 -456.8,E2 -456.8} C_VEL
LIN {X 0,Y 608.456,Z 375.982,A -85,B 0,C 180,E1 -457.801,E2 -457.801} C_VEL
LIN {X 0,Y 608.472,Z 367.527,A -85,B 0,C 180,E1 -458.637,E2 -458.637} C_VEL
LIN {X 0,Y 608.481,Z 357.08,A -85,B 0,C 180,E1 -459.474,E2 -459.474} C_VEL
LIN {X 0,Y 608.489,Z 346.743,A -85,B 0,C 180,E1 -460.146,E2 -460.146} C_VEL
LIN {X 0,Y 608.515,Z 335.595,A -85,B 0,C 180,E1 -460.725,E2 -460.725} C_VEL
LIN {X 0,Y 608.522,Z 323.886,A -85,B 0,C 180,E1 -461.192,E2 -461.192} C_VEL
LIN {X 0,Y 608.546,Z 311.234,A -85,B 0,C 180,E1 -461.555,E2 -461.555} C_VEL
LIN {X 0,Y 608.573,Z 298.547,A -85,B 0,C 180,E1 -461.787,E2 -461.787} C_VEL
LIN {X 0,Y 608.494,Z 294.902,A -85,B 0,C 180,E1 -461.852,E2 -461.852} C_VEL
LIN {X 0,Y 608.484,Z 273.794,A -85,B 0,C 180,E1 -464.55,E2 -464.55} C_VEL
LIN {X 0,Y 608.518,Z 252.521,A -85,B 0,C 180,E1 -467.302,E2 -467.302} C_VEL
LIN {X 0,Y 608.557,Z 231.247,A -85,B 0,C 180,E1 -470.095,E2 -470.095} C_VEL
LIN {X 0,Y 608.583,Z 211.306,A -85,B 0,C 180,E1 -472.76,E2 -472.76} C_VEL
LIN {X 0,Y 608.648,Z 190.183,A -85,B 0,C 180,E1 -475.638,E2 -475.638} C_VEL
LIN {X 0,Y 608.681,Z 171.415,A -85,B 0,C 180,E1 -478.256,E2 -478.256} C_VEL
LIN {X 0,Y 608.433,Z 167.694,A -85,B 0,C 180,E1 -478.813,E2 -478.813} C_VEL
LIN {X 0,Y 608.446,Z 167.698,A -85,B 0,C 180,E1 -481.318,E2 -481.318} C_VEL
LIN {X 0,Y 608.428,Z 167.694,A -85,B 0,C 180,E1 -483.728,E2 -483.728} C_VEL
LIN {X 0,Y 608.432,Z 167.693,A -85,B 0,C 180,E1 -486.094,E2 -486.094} C_VEL
LIN {X 0,Y 608.436,Z 167.699,A -85,B 0,C 180,E1 -488.591,E2 -488.591} C_VEL
LIN {X 0,Y 608.45,Z 167.69,A -85,B 0,C 180,E1 -491.341,E2 -491.341} C_VEL
LIN {X 0,Y 608.453,Z 167.692,A -85,B 0,C 180,E1 -494.263,E2 -494.263} C_VEL
LIN {X 0,Y 608.455,Z 167.693,A -85,B 0,C 180,E1 -497.04,E2 -497.04} C_VEL
LIN {X 0,Y 608.425,Z 167.694,A -85,B 0,C 180,E1 -499.694,E2 -499.694} C_VEL
LIN {X 0,Y 608.445,Z 167.693,A -85,B 0,C 180,E1 -502.252,E2 -502.252} C_VEL
LIN {X 0,Y 608.401,Z 167.697,A -85,B 0,C 180,E1 -505.102,E2 -505.102} C_VEL
LIN {X 0,Y 608.429,Z 167.899,A -85,B 0,C 180,E1 -505.929,E2 -505.929} C_VEL
LIN {X 0,Y 608.46,Z 176.716,A -85,B 0,C 180,E1 -508.295,E2 -508.295} C_VEL
LIN {X 0,Y 608.431,Z 185.965,A -85,B 0,C 180,E1 -510.978,E2 -510.978} C_VEL
LIN {X 0,Y 608.45,Z 192.843,A -85,B 0,C 180,E1 -513.226,E2 -513.226} C_VEL
LIN {X 0,Y 608.479,Z 200.8,A -85,B 0,C 180,E1 -515.848,E2 -515.848} C_VEL
LIN {X 0,Y 608.444,Z 209.533,A -85,B 0,C 180,E1 -518.663,E2 -518.663} C_VEL
LIN {X 0,Y 608.449,Z 217.835,A -85,B 0,C 180,E1 -521.291,E2 -521.291} C_VEL
LIN {X 0,Y 608.443,Z 226.224,A -85,B 0,C 180,E1 -523.906,E2 -523.906} C_VEL
LIN {X 0,Y 608.437,Z 235.127,A -85,B 0,C 180,E1 -526.643,E2 -526.643} C_VEL
LIN {X 0,Y 608.445,Z 240.663,A -85,B 0,C 180,E1 -528.285,E2 -528.285} C_VEL
LIN {X 0,Y 608.531,Z 253.824,A -85,B 0,C 180,E1 -528.551,E2 -528.551} C_VEL
LIN {X 0,Y 608.508,Z 266.454,A -85,B 0,C 180,E1 -528.945,E2 -528.945} C_VEL
LIN {X 0,Y 608.501,Z 277.987,A -85,B 0,C 180,E1 -529.435,E2 -529.435} C_VEL
LIN {X 0,Y 608.488,Z 290.221,A -85,B 0,C 180,E1 -530.107,E2 -530.107} C_VEL
LIN {X 0,Y 608.472,Z 300.965,A -85,B 0,C 180,E1 -530.862,E2 -530.862} C_VEL
LIN {X 0,Y 608.475,Z 310.635,A -85,B 0,C 180,E1 -531.699,E2 -531.699} C_VEL
LIN {X 0,Y 608.47,Z 318.565,A -85,B 0,C 180,E1 -532.534,E2 -532.534} C_VEL
LIN {X 0,Y 608.468,Z 326.071,A -85,B 0,C 180,E1 -533.497,E2 -533.497} C_VEL
LIN {X 0,Y 608.451,Z 331.609,A -85,B 0,C 180,E1 -534.366,E2 -534.366} C_VEL
LIN {X 0,Y 608.43,Z 336.751,A -85,B 0,C 180,E1 -535.362,E2 -535.362} C_VEL
LIN {X 0,Y 608.448,Z 340.741,A -85,B 0,C 180,E1 -536.358,E2 -536.358} C_VEL
LIN {X 0,Y 608.425,Z 343.691,A -85,B 0,C 180,E1 -537.352,E2 -537.352} C_VEL
LIN {X 0,Y 608.442,Z 345.127,A -85,B 0,C 180,E1 -538.014,E2 -538.014} C_VEL
LIN {X 0,Y 608.44,Z 346.752,A -85,B 0,C 180,E1 -539.338,E2 -539.338} C_VEL
LIN {X 0,Y 608.434,Z 346.995,A -85,B 0,C 180,E1 -540,E2 -540} C_VEL
LIN {X 0,Y 608.438,Z 346.815,A -85,B 0,C 180,E1 -540.662,E2 -540.662} C_VEL
LIN {X 0,Y 608.441,Z 345.276,A -85,B 0,C 180,E1 -541.986,E2 -541.986} C_VEL
LIN {X 0,Y 608.426,Z 343.918,A -85,B 0,C 180,E1 -542.648,E2 -542.648} C_VEL
LIN {X 0,Y 608.45,Z 341.042,A -85,B 0,C 180,E1 -543.642,E2 -543.642} C_VEL
LIN {X 0,Y 608.433,Z 337.143,A -85,B 0,C 180,E1 -544.638,E2 -544.638} C_VEL
LIN {X 0,Y 608.45,Z 332.113,A -85,B 0,C 180,E1 -545.634,E2 -545.634} C_VEL
LIN {X 0,Y 608.441,Z 325.794,A -85,B 0,C 180,E1 -546.633,E2 -546.633} C_VEL
LIN {X 0,Y 608.476,Z 317.879,A -85,B 0,C 180,E1 -547.633,E2 -547.633} C_VEL
LIN {X 0,Y 608.472,Z 308.034,A -85,B 0,C 180,E1 -548.636,E2 -548.636} C_VEL
LIN {X 0,Y 608.477,Z 305.938,A -85,B 0,C 180,E1 -548.819,E2 -548.819} C_VEL
LIN {X 0,Y 607.8,Z 301.604,A -85,B 0,C 180,E1 -549.19,E2 -549.19} C_VEL
LIN {X 0,Y 604.923,Z 294.362,A -85,B 0,C 180,E1 -549.769,E2 -549.769} C_VEL
LIN {X 0,Y 602.09,Z 286.725,A -85,B 0,C 180,E1 -550.301,E2 -550.301} C_VEL
LIN {X 0,Y 601.483,Z 281.659,A -85,B 0,C 180,E1 -550.594,E2 -550.594} C_VEL
LIN {X 0,Y 601.525,Z 270.151,A -85,B 0,C 180,E1 -551.133,E2 -551.133} C_VEL
LIN {X 0,Y 601.594,Z 257.068,A -85,B 0,C 180,E1 -551.583,E2 -551.583} C_VEL
LIN {X 0,Y 601.589,Z 244.231,A -85,B 0,C 180,E1 -551.882,E2 -551.882} C_VEL
LIN {X 0,Y 601.328,Z 240.499,A -85,B 0,C 180,E1 -551.952,E2 -551.952} C_VEL
LIN {X 0,Y 601.323,Z 233.193,A -85,B 0,C 180,E1 -554.208,E2 -554.208} C_VEL
LIN {X 0,Y 601.368,Z 224.286,A -85,B 0,C 180,E1 -556.988,E2 -556.988} C_VEL
LIN {X 0,Y 601.364,Z 215.38,A -85,B 0,C 180,E1 -559.811,E2 -559.811} C_VEL
LIN {X 0,Y 601.412,Z 206.472,A -85,B 0,C 180,E1 -562.683,E2 -562.683} C_VEL
LIN {X 0,Y 601.391,Z 197.565,A -85,B 0,C 180,E1 -565.62,E2 -565.62} C_VEL
LIN {X 0,Y 601.434,Z 189.742,A -85,B 0,C 180,E1 -568.246,E2 -568.246} C_VEL
LIN {X 0,Y 601.467,Z 181.437,A -85,B 0,C 180,E1 -570.939,E2 -570.939} C_VEL
LIN {X 0,Y 601.447,Z 174.122,A -85,B 0,C 180,E1 -573.312,E2 -573.312} C_VEL
LIN {X 0,Y 601.385,Z 168.575,A -85,B 0,C 180,E1 -575.11,E2 -575.11} C_VEL
LIN {X 0,Y 601.405,Z 168.571,A -85,B 0,C 180,E1 -577.421,E2 -577.421} C_VEL
LIN {X 0,Y 601.405,Z 168.57,A -85,B 0,C 180,E1 -579.996,E2 -579.996} C_VEL
LIN {X 0,Y 601.41,Z 168.575,A -85,B 0,C 180,E1 -582.671,E2 -582.671} C_VEL
LIN {X 0,Y 601.404,Z 168.571,A -85,B 0,C 180,E1 -585.479,E2 -585.479} C_VEL
LIN {X 0,Y 601.426,Z 168.566,A -85,B 0,C 180,E1 -588.407,E2 -588.407} C_VEL
LIN {X 0,Y 601.406,Z 168.574,A -85,B 0,C 180,E1 -590.872,E2 -590.872} C_VEL
LIN {X 0,Y 601.391,Z 168.575,A -85,B 0,C 180,E1 -593.741,E2 -593.741} C_VEL
LIN {X 0,Y 601.417,Z 168.569,A -85,B 0,C 180,E1 -596.685,E2 -596.685} C_VEL
LIN {X 0,Y 601.418,Z 168.57,A -85,B 0,C 180,E1 -599.057,E2 -599.057} C_VEL
LIN {X 0,Y 601.391,Z 168.872,A -85,B 0,C 180,E1 -600.605,E2 -600.605} C_VEL
LIN {X 0,Y 601.385,Z 172.094,A -85,B 0,C 180,E1 -602.885,E2 -602.885} C_VEL
LIN {X 0,Y 601.344,Z 175.168,A -85,B 0,C 180,E1 -605.118,E2 -605.118} C_VEL
LIN {X 0,Y 601.337,Z 178.509,A -85,B 0,C 180,E1 -607.413,E2 -607.413} C_VEL
LIN {X 0,Y 601.31,Z 182.762,A -85,B 0,C 180,E1 -610.187,E2 -610.187} C_VEL
LIN {X 0,Y 601.327,Z 187.168,A -85,B 0,C 180,E1 -613.01,E2 -613.01} C_VEL
LIN {X 0,Y 601.337,Z 191.813,A -85,B 0,C 180,E1 -615.942,E2 -615.942} C_VEL
LIN {X 0,Y 601.325,Z 196.786,A -85,B 0,C 180,E1 -619.039,E2 -619.039} C_VEL
LIN {X 0,Y 601.292,Z 201.486,A -85,B 0,C 180,E1 -621.936,E2 -621.936} C_VEL
LIN {X 0,Y 601.334,Z 203.447,A -85,B 0,C 180,E1 -623.139,E2 -623.139} C_VEL
LIN {X 0,Y 601.365,Z 213.525,A -85,B 0,C 180,E1 -623.522,E2 -623.522} C_VEL
LIN {X 0,Y 601.336,Z 221.948,A -85,B 0,C 180,E1 -623.961,E2 -623.961} C_VEL
LIN {X 0,Y 601.323,Z 230.276,A -85,B 0,C 180,E1 -624.55,E2 -624.55} C_VEL
LIN {X 0,Y 601.394,Z 236.733,A -85,B 0,C 180,E1 -625.139,E2 -625.139} C_VEL
LIN {X 0,Y 601.349,Z 242.556,A -85,B 0,C 180,E1 -625.81,E2 -625.81} C_VEL
LIN {X 0,Y 601.35,Z 248.018,A -85,B 0,C 180,E1 -626.649,E2 -626.649} C_VEL
LIN {X 0,Y 601.331,Z 251.341,A -85,B 0,C 180,E1 -627.32,E2 -627.32} C_VEL
LIN {X 0,Y 601.343,Z 253.829,A -85,B 0,C 180,E1 -627.99,E2 -627.99} C_VEL
LIN {X 0,Y 601.348,Z 255.566,A -85,B 0,C 180,E1 -628.66,E2 -628.66} C_VEL
LIN {X 0,Y 601.34,Z 256.606,A -85,B 0,C 180,E1 -629.329,E2 -629.329} C_VEL
LIN {X 0,Y 601.335,Z 256.988,A -85,B 0,C 180,E1 -629.999,E2 -629.999} C_VEL
LIN {X 0,Y 601.339,Z 256.711,A -85,B 0,C 180,E1 -630.669,E2 -630.669} C_VEL
LIN {X 0,Y 601.349,Z 255.769,A -85,B 0,C 180,E1 -631.338,E2 -631.338} C_VEL
LIN {X 0,Y 601.342,Z 254.131,A -85,B 0,C 180,E1 -632.008,E2 -632.008} C_VEL
LIN {X 0,Y 601.332,Z 251.751,A -85,B 0,C 180,E1 -632.679,E2 -632.679} C_VEL
LIN {X 0,Y 601.375,Z 246.626,A -85,B 0,C 180,E1 -633.684,E2 -633.684} C_VEL
LIN {X 0,Y 601.378,Z 240.559,A -85,B 0,C 180,E1 -634.524,E2 -634.524} C_VEL
LIN {X 0,Y 601.356,Z 234.258,A -85,B 0,C 180,E1 -635.196,E2 -635.196} C_VEL
LIN {X 0,Y 601.32,Z 227.099,A -85,B 0,C 180,E1 -635.785,E2 -635.785} C_VEL
LIN {X 0,Y 601.333,Z 219.123,A -85,B 0,C 180,E1 -636.289,E2 -636.289} C_VEL
LIN {X 0,Y 601.412,Z 210.257,A -85,B 0,C 180,E1 -636.71,E2 -636.71} C_VEL
LIN {X 0,Y 601.338,Z 203.438,A -85,B 0,C 180,E1 -636.956,E2 -636.956} C_VEL
LIN {X 0,Y 601.289,Z 199.432,A -85,B 0,C 180,E1 -639.417,E2 -639.417} C_VEL
LIN {X 0,Y 601.315,Z 195.025,A -85,B 0,C 180,E1 -642.144,E2 -642.144} C_VEL
LIN {X 0,Y 601.297,Z 190.618,A -85,B 0,C 180,E1 -644.899,E2 -644.899} C_VEL
LIN {X 0,Y 601.322,Z 187.312,A -85,B 0,C 180,E1 -646.988,E2 -646.988} C_VEL
LIN {X 0,Y 601.307,Z 182.904,A -85,B 0,C 180,E1 -649.812,E2 -649.812} C_VEL
LIN {X 0,Y 601.331,Z 178.648,A -85,B 0,C 180,E1 -652.585,E2 -652.585} C_VEL
LIN {X 0,Y 601.34,Z 175.314,A -85,B 0,C 180,E1 -654.88,E2 -654.88} C_VEL
LIN {X 0,Y 601.392,Z 171.865,A -85,B 0,C 180,E1 -657.358,E2 -657.358} C_VEL
LIN {X 0,Y 601.382,Z 168.986,A -85,B 0,C 180,E1 -659.394,E2 -659.394} C_VEL
LIN {X 0,Y 601.425,Z 168.567,A -85,B 0,C 180,E1 -660.163,E2 -660.163} C_VEL
LIN {X 0,Y 601.405,Z 168.566,A -85,B 0,C 180,E1 -662.712,E2 -662.712} C_VEL
LIN {X 0,Y 601.382,Z 168.573,A -85,B 0,C 180,E1 -665.11,E2 -665.11} C_VEL
LIN {X 0,Y 601.429,Z 168.573,A -85,B 0,C 180,E1 -667.418,E2 -667.418} C_VEL
LIN {X 0,Y 601.406,Z 168.567,A -85,B 0,C 180,E1 -669.994,E2 -669.994} C_VEL
LIN {X 0,Y 601.402,Z 168.569,A -85,B 0,C 180,E1 -672.669,E2 -672.669} C_VEL
LIN {X 0,Y 601.419,Z 168.567,A -85,B 0,C 180,E1 -675.481,E2 -675.481} C_VEL
LIN {X 0,Y 601.417,Z 168.567,A -85,B 0,C 180,E1 -678.406,E2 -678.406} C_VEL
LIN {X 0,Y 601.431,Z 168.571,A -85,B 0,C 180,E1 -680.875,E2 -680.875} C_VEL
LIN {X 0,Y 601.436,Z 168.562,A -85,B 0,C 180,E1 -683.733,E2 -683.733} C_VEL
LIN {X 0,Y 601.426,Z 168.57,A -85,B 0,C 180,E1 -686.686,E2 -686.686} C_VEL
LIN {X 0,Y 601.423,Z 168.565,A -85,B 0,C 180,E1 -689.058,E2 -689.058} C_VEL
LIN {X 0,Y 601.431,Z 168.563,A -85,B 0,C 180,E1 -691.373,E2 -691.373} C_VEL
LIN {X 0,Y 601.412,Z 168.575,A -85,B 0,C 180,E1 -694.13,E2 -694.13} C_VEL
LIN {X 0,Y 601.417,Z 168.567,A -85,B 0,C 180,E1 -696.589,E2 -696.589} C_VEL
LIN {X 0,Y 601.429,Z 168.566,A -85,B 0,C 180,E1 -699.478,E2 -699.478} C_VEL
LIN {X 0,Y 601.387,Z 168.57,A -85,B 0,C 180,E1 -702.311,E2 -702.311} C_VEL
LIN {X 0,Y 601.409,Z 168.566,A -85,B 0,C 180,E1 -704.408,E2 -704.408} C_VEL
LIN {X 0,Y 601.42,Z 168.568,A -85,B 0,C 180,E1 -707.172,E2 -707.172} C_VEL
LIN {X 0,Y 601.418,Z 168.567,A -85,B 0,C 180,E1 -709.905,E2 -709.905} C_VEL
LIN {X 0,Y 601.444,Z 168.562,A -85,B 0,C 180,E1 -712.615,E2 -712.615} C_VEL
LIN {X 0,Y 601.415,Z 168.572,A -85,B 0,C 180,E1 -715.308,E2 -715.308} C_VEL
LIN {X 0,Y 601.399,Z 168.567,A -85,B 0,C 180,E1 -717.991,E2 -717.991} C_VEL
LIN {X 0,Y 601.455,Z 168.565,A -85,B 0,C 180,E1 -720.669,E2 -720.669} C_VEL
LIN {X 0,Y 601.402,Z 168.568,A -85,B 0,C 180,E1 -723.35,E2 -723.35} C_VEL
LIN {X 0,Y 601.388,Z 168.569,A -85,B 0,C 180,E1 -726.037,E2 -726.037} C_VEL
LIN {X 0,Y 601.428,Z 168.57,A -85,B 0,C 180,E1 -728.738,E2 -728.738} C_VEL
LIN {X 0,Y 601.39,Z 168.568,A -85,B 0,C 180,E1 -731.459,E2 -731.459} C_VEL
LIN {X 0,Y 601.406,Z 168.574,A -85,B 0,C 180,E1 -734.206,E2 -734.206} C_VEL
LIN {X 0,Y 601.388,Z 168.568,A -85,B 0,C 180,E1 -736.987,E2 -736.987} C_VEL
LIN {X 0,Y 601.379,Z 168.575,A -85,B 0,C 180,E1 -739.81,E2 -739.81} C_VEL
LIN {X 0,Y 601.385,Z 168.569,A -85,B 0,C 180,E1 -742.684,E2 -742.684} C_VEL
LIN {X 0,Y 601.361,Z 168.571,A -85,B 0,C 180,E1 -744.88,E2 -744.88} C_VEL
LIN {X 0,Y 601.368,Z 168.575,A -85,B 0,C 180,E1 -747.356,E2 -747.356} C_VEL
LIN {X 0,Y 601.388,Z 168.57,A -85,B 0,C 180,E1 -750.166,E2 -750.166} C_VEL
LIN {X 0,Y 601.381,Z 168.57,A -85,B 0,C 180,E1 -752.712,E2 -752.712} C_VEL
LIN {X 0,Y 601.369,Z 168.576,A -85,B 0,C 180,E1 -755.111,E2 -755.111} C_VEL
LIN {X 0,Y 601.422,Z 168.571,A -85,B 0,C 180,E1 -757.42,E2 -757.42} C_VEL
LIN {X 0,Y 601.369,Z 168.57,A -85,B 0,C 180,E1 -759.999,E2 -759.999} C_VEL
LIN {X 0,Y 601.378,Z 168.574,A -85,B 0,C 180,E1 -762.673,E2 -762.673} C_VEL
LIN {X 0,Y 601.39,Z 168.57,A -85,B 0,C 180,E1 -765.48,E2 -765.48} C_VEL
LIN {X 0,Y 601.412,Z 168.569,A -85,B 0,C 180,E1 -768.408,E2 -768.408} C_VEL
LIN {X 0,Y 601.425,Z 168.57,A -85,B 0,C 180,E1 -770.876,E2 -770.876} C_VEL
LIN {X 0,Y 601.398,Z 168.567,A -85,B 0,C 180,E1 -773.418,E2 -773.418} C_VEL
LIN {X 0,Y 601.427,Z 168.568,A -85,B 0,C 180,E1 -776.065,E2 -776.065} C_VEL
LIN {X 0,Y 601.416,Z 168.566,A -85,B 0,C 180,E1 -779.059,E2 -779.059} C_VEL
LIN {X 0,Y 601.431,Z 168.653,A -85,B 0,C 180,E1 -780.97,E2 -780.97} C_VEL
LIN {X 0,Y 601.899,Z 172.761,A -85,B 0,C 180,E1 -781.589,E2 -781.589} C_VEL
LIN {X 0,Y 601.814,Z 192.703,A -85,B 0,C 180,E1 -784.401,E2 -784.401} C_VEL
LIN {X 0,Y 601.702,Z 214.853,A -85,B 0,C 180,E1 -787.449,E2 -787.449} C_VEL
LIN {X 0,Y 601.601,Z 235.25,A -85,B 0,C 180,E1 -790.198,E2 -790.198} C_VEL
LIN {X 0,Y 601.543,Z 257.765,A -85,B 0,C 180,E1 -793.182,E2 -793.182} C_VEL
LIN {X 0,Y 601.478,Z 280.776,A -85,B 0,C 180,E1 -796.184,E2 -796.184} C_VEL
LIN {X 0,Y 601.442,Z 294.915,A -85,B 0,C 180,E1 -798.009,E2 -798.009} C_VEL
LIN {X 0,Y 601.578,Z 310.394,A -85,B 0,C 180,E1 -798.289,E2 -798.289} C_VEL
LIN {X 0,Y 601.551,Z 323.426,A -85,B 0,C 180,E1 -798.661,E2 -798.661} C_VEL
LIN {X 0,Y 601.542,Z 335.611,A -85,B 0,C 180,E1 -799.15,E2 -799.15} C_VEL
LIN {X 0,Y 601.468,Z 346.774,A -85,B 0,C 180,E1 -799.737,E2 -799.737} C_VEL
LIN {X 0,Y 601.462,Z 358.267,A -85,B 0,C 180,E1 -800.501,E2 -800.501} C_VEL
LIN {X 0,Y 601.436,Z 367.547,A -85,B 0,C 180,E1 -801.263,E2 -801.263} C_VEL
LIN {X 0,Y 601.4,Z 375.998,A -85,B 0,C 180,E1 -802.109,E2 -802.109} C_VEL
LIN {X 0,Y 601.387,Z 384.242,A -85,B 0,C 180,E1 -803.121,E2 -803.121} C_VEL
LIN {X 0,Y 601.373,Z 390.883,A -85,B 0,C 180,E1 -804.132,E2 -804.132} C_VEL
LIN {X 0,Y 601.336,Z 396.954,A -85,B 0,C 180,E1 -805.308,E2 -805.308} C_VEL
LIN {X 0,Y 601.368,Z 400.899,A -85,B 0,C 180,E1 -806.316,E2 -806.316} C_VEL
LIN {X 0,Y 601.325,Z 403.812,A -85,B 0,C 180,E1 -807.321,E2 -807.321} C_VEL
LIN {X 0,Y 601.343,Z 405.203,A -85,B 0,C 180,E1 -807.992,E2 -807.992} C_VEL
LIN {X 0,Y 601.339,Z 406.784,A -85,B 0,C 180,E1 -809.331,E2 -809.331} C_VEL
LIN {X 0,Y 601.335,Z 407,A -85,B 0,C 180,E1 -810.001,E2 -810.001} C_VEL
LIN {X 0,Y 601.347,Z 406.183,A -85,B 0,C 180,E1 -811.34,E2 -811.34} C_VEL
LIN {X 0,Y 601.343,Z 405.2,A -85,B 0,C 180,E1 -812.01,E2 -812.01} C_VEL
LIN {X 0,Y 601.325,Z 403.807,A -85,B 0,C 180,E1 -812.68,E2 -812.68} C_VEL
LIN {X 0,Y 601.368,Z 400.893,A -85,B 0,C 180,E1 -813.686,E2 -813.686} C_VEL
LIN {X 0,Y 601.336,Z 396.946,A -85,B 0,C 180,E1 -814.693,E2 -814.693} C_VEL
LIN {X 0,Y 601.373,Z 390.872,A -85,B 0,C 180,E1 -815.87,E2 -815.87} C_VEL
LIN {X 0,Y 601.382,Z 384.23,A -85,B 0,C 180,E1 -816.881,E2 -816.881} C_VEL
LIN {X 0,Y 601.401,Z 375.982,A -85,B 0,C 180,E1 -817.893,E2 -817.893} C_VEL
LIN {X 0,Y 601.436,Z 367.528,A -85,B 0,C 180,E1 -818.738,E2 -818.738} C_VEL
LIN {X 0,Y 601.449,Z 357.082,A -85,B 0,C 180,E1 -819.586,E2 -819.586} C_VEL
LIN {X 0,Y 601.469,Z 346.744,A -85,B 0,C 180,E1 -820.265,E2 -820.265} C_VEL
LIN {X 0,Y 601.539,Z 334.581,A -85,B 0,C 180,E1 -820.897,E2 -820.897} C_VEL
LIN {X 0,Y 601.557,Z 322.196,A -85,B 0,C 180,E1 -821.379,E2 -821.379} C_VEL
LIN {X 0,Y 601.585,Z 309.406,A -85,B 0,C 180,E1 -821.734,E2 -821.734} C_VEL
LIN {X 0,Y 601.573,Z 296.139,A -85,B 0,C 180,E1 -821.958,E2 -821.958} C_VEL
LIN {X 0,Y 601.443,Z 294.902,A -85,B 0,C 180,E1 -821.993,E2 -821.993} C_VEL
LIN {X 0,Y 601.469,Z 273.794,A -85,B 0,C 180,E1 -824.724,E2 -824.724} C_VEL
LIN {X 0,Y 601.541,Z 252.521,A -85,B 0,C 180,E1 -827.509,E2 -827.509} C_VEL
LIN {X 0,Y 601.613,Z 232.577,A -85,B 0,C 180,E1 -830.159,E2 -830.159} C_VEL
LIN {X 0,Y 601.686,Z 212.633,A -85,B 0,C 180,E1 -832.854,E2 -832.854} C_VEL
LIN {X 0,Y 601.81,Z 192.689,A -85,B 0,C 180,E1 -835.601,E2 -835.601} C_VEL
LIN {X 0,Y 601.895,Z 174.105,A -85,B 0,C 180,E1 -838.223,E2 -838.223} C_VEL
LIN {X 0,Y 601.721,Z 169.933,A -85,B 0,C 180,E1 -838.838,E2 -838.838} C_VEL
LIN {X 0,Y 601.394,Z 168.575,A -85,B 0,C 180,E1 -839.06,E2 -839.06} C_VEL
LIN {X 0,Y 601.387,Z 168.574,A -85,B 0,C 180,E1 -841.728,E2 -841.728} C_VEL
LIN {X 0,Y 601.403,Z 168.568,A -85,B 0,C 180,E1 -844.121,E2 -844.121} C_VEL
LIN {X 0,Y 601.434,Z 168.565,A -85,B 0,C 180,E1 -847.382,E2 -847.382} C_VEL
LIN {X 0,Y 601.402,Z 168.572,A -85,B 0,C 180,E1 -849.996,E2 -849.996} C_VEL
LIN {X 0,Y 601.413,Z 168.567,A -85,B 0,C 180,E1 -852.671,E2 -852.671} C_VEL
LIN {X 0,Y 601.403,Z 168.574,A -85,B 0,C 180,E1 -855.48,E2 -855.48} C_VEL
LIN {X 0,Y 601.423,Z 168.566,A -85,B 0,C 180,E1 -858.408,E2 -858.408} C_VEL
LIN {X 0,Y 601.405,Z 168.576,A -85,B 0,C 180,E1 -860.873,E2 -860.873} C_VEL
LIN {X 0,Y 601.381,Z 168.571,A -85,B 0,C 180,E1 -863.415,E2 -863.415} C_VEL
LIN {X 0,Y 601.362,Z 168.679,A -85,B 0,C 180,E1 -865.972,E2 -865.972} C_VEL
LIN {X 0,Y 601.391,Z 177.265,A -85,B 0,C 180,E1 -868.272,E2 -868.272} C_VEL
LIN {X 0,Y 601.389,Z 185.372,A -85,B 0,C 180,E1 -870.605,E2 -870.605} C_VEL
LIN {X 0,Y 601.441,Z 192.82,A -85,B 0,C 180,E1 -872.888,E2 -872.888} C_VEL
LIN {X 0,Y 601.457,Z 201.746,A -85,B 0,C 180,E1 -875.86,E2 -875.86} C_VEL
LIN {X 0,Y 601.405,Z 210.647,A -85,B 0,C 180,E1 -878.761,E2 -878.761} C_VEL
LIN {X 0,Y 601.399,Z 219.549,A -85,B 0,C 180,E1 -881.607,E2 -881.607} C_VEL
LIN {X 0,Y 601.37,Z 228.452,A -85,B 0,C 180,E1 -884.408,E2 -884.408} C_VEL
LIN {X 0,Y 601.385,Z 236.242,A -85,B 0,C 180,E1 -886.827,E2 -886.827} C_VEL
LIN {X 0,Y 601.403,Z 240.702,A -85,B 0,C 180,E1 -888.146,E2 -888.146} C_VEL
LIN {X 0,Y 601.598,Z 253.002,A -85,B 0,C 180,E1 -888.396,E2 -888.396} C_VEL
LIN {X 0,Y 601.543,Z 265.54,A -85,B 0,C 180,E1 -888.78,E2 -888.78} C_VEL
LIN {X 0,Y 601.514,Z 278.002,A -85,B 0,C 180,E1 -889.311,E2 -889.311} C_VEL
LIN {X 0,Y 601.479,Z 290.23,A -85,B 0,C 180,E1 -889.991,E2 -889.991} C_VEL
LIN {X 0,Y 601.433,Z 300.973,A -85,B 0,C 180,E1 -890.754,E2 -890.754} C_VEL
LIN {X 0,Y 601.429,Z 310.642,A -85,B 0,C 180,E1 -891.601,E2 -891.601} C_VEL
LIN {X 0,Y 601.418,Z 318.571,A -85,B 0,C 180,E1 -892.446,E2 -892.446} C_VEL
LIN {X 0,Y 601.377,Z 325.886,A -85,B 0,C 180,E1 -893.393,E2 -893.393} C_VEL
LIN {X 0,Y 601.372,Z 331.61,A -85,B 0,C 180,E1 -894.299,E2 -894.299} C_VEL
LIN {X 0,Y 601.335,Z 336.751,A -85,B 0,C 180,E1 -895.307,E2 -895.307} C_VEL
LIN {X 0,Y 601.367,Z 340.74,A -85,B 0,C 180,E1 -896.315,E2 -896.315} C_VEL
LIN {X 0,Y 601.324,Z 343.693,A -85,B 0,C 180,E1 -897.32,E2 -897.32} C_VEL
LIN {X 0,Y 601.341,Z 345.128,A -85,B 0,C 180,E1 -897.991,E2 -897.991} C_VEL
LIN {X 0,Y 601.34,Z 346.753,A -85,B 0,C 180,E1 -899.33,E2 -899.33} C_VEL
LIN {X 0,Y 601.335,Z 346.996,A -85,B 0,C 180,E1 -900,E2 -900} C_VEL
LIN {X 0,Y 601.339,Z 346.815,A -85,B 0,C 180,E1 -900.67,E2 -900.67} C_VEL
LIN {X 0,Y 601.34,Z 345.276,A -85,B 0,C 180,E1 -902.009,E2 -902.009} C_VEL
LIN {X 0,Y 601.326,Z 343.917,A -85,B 0,C 180,E1 -902.68,E2 -902.68} C_VEL
LIN {X 0,Y 601.368,Z 341.043,A -85,B 0,C 180,E1 -903.685,E2 -903.685} C_VEL
LIN {X 0,Y 601.337,Z 337.144,A -85,B 0,C 180,E1 -904.693,E2 -904.693} C_VEL
LIN {X 0,Y 601.373,Z 332.113,A -85,B 0,C 180,E1 -905.701,E2 -905.701} C_VEL
LIN {X 0,Y 601.383,Z 325.787,A -85,B 0,C 180,E1 -906.711,E2 -906.711} C_VEL
LIN {X 0,Y 601.396,Z 317.876,A -85,B 0,C 180,E1 -907.723,E2 -907.723} C_VEL
LIN {X 0,Y 601.437,Z 308.025,A -85,B 0,C 180,E1 -908.738,E2 -908.738} C_VEL
LIN {X 0,Y 601.447,Z 297.707,A -85,B 0,C 180,E1 -909.585,E2 -909.585} C_VEL
LIN {X 0,Y 601.449,Z 286.089,A -85,B 0,C 180,E1 -910.35,E2 -910.35} C_VEL
LIN {X 0,Y 601.483,Z 281.659,A -85,B 0,C 180,E1 -910.594,E2 -910.594} C_VEL
LIN {X 0,Y 600.879,Z 276.526,A -85,B 0,C 180,E1 -910.869,E2 -910.869} C_VEL
LIN {X 0,Y 598.07,Z 268.078,A -85,B 0,C 180,E1 -911.291,E2 -911.291} C_VEL
LIN {X 0,Y 595.256,Z 259.328,A -85,B 0,C 180,E1 -911.646,E2 -911.646} C_VEL
LIN {X 0,Y 594.637,Z 253.728,A -85,B 0,C 180,E1 -911.814,E2 -911.814} C_VEL
LIN {X 0,Y 594.449,Z 241.912,A -85,B 0,C 180,E1 -912.066,E2 -912.066} C_VEL
LIN {X 0,Y 594.246,Z 240.427,A -85,B 0,C 180,E1 -912.118,E2 -912.118} C_VEL
LIN {X 0,Y 594.288,Z 232.078,A -85,B 0,C 180,E1 -914.73,E2 -914.73} C_VEL
LIN {X 0,Y 594.297,Z 223.171,A -85,B 0,C 180,E1 -917.551,E2 -917.551} C_VEL
LIN {X 0,Y 594.326,Z 214.264,A -85,B 0,C 180,E1 -920.417,E2 -920.417} C_VEL
LIN {X 0,Y 594.336,Z 205.357,A -85,B 0,C 180,E1 -923.337,E2 -923.337} C_VEL
LIN {X 0,Y 594.37,Z 197.335,A -85,B 0,C 180,E1 -926.019,E2 -926.019} C_VEL
LIN {X 0,Y 594.425,Z 189.63,A -85,B 0,C 180,E1 -928.589,E2 -928.589} C_VEL
LIN {X 0,Y 594.417,Z 181.197,A -85,B 0,C 180,E1 -931.348,E2 -931.348} C_VEL
LIN {X 0,Y 594.39,Z 173.767,A -85,B 0,C 180,E1 -933.761,E2 -933.761} C_VEL
LIN {X 0,Y 594.349,Z 169.451,A -85,B 0,C 180,E1 -935.197,E2 -935.197} C_VEL
LIN {X 0,Y 594.378,Z 169.451,A -85,B 0,C 180,E1 -937.942,E2 -937.942} C_VEL
LIN {X 0,Y 594.379,Z 169.448,A -85,B 0,C 180,E1 -940.821,E2 -940.821} C_VEL
LIN {X 0,Y 594.353,Z 169.448,A -85,B 0,C 180,E1 -943.301,E2 -943.301} C_VEL
LIN {X 0,Y 594.365,Z 169.449,A -85,B 0,C 180,E1 -946.161,E2 -946.161} C_VEL
LIN {X 0,Y 594.383,Z 169.444,A -85,B 0,C 180,E1 -948.536,E2 -948.536} C_VEL
LIN {X 0,Y 594.374,Z 169.446,A -85,B 0,C 180,E1 -951.297,E2 -951.297} C_VEL
LIN {X 0,Y 594.346,Z 169.453,A -85,B 0,C 180,E1 -953.754,E2 -953.754} C_VEL
LIN {X 0,Y 594.368,Z 169.446,A -85,B 0,C 180,E1 -956.237,E2 -956.237} C_VEL
LIN {X 0,Y 594.375,Z 169.45,A -85,B 0,C 180,E1 -958.649,E2 -958.649} C_VEL
LIN {X 0,Y 594.34,Z 169.454,A -85,B 0,C 180,E1 -960.221,E2 -960.221} C_VEL
LIN {X 0,Y 594.306,Z 170.247,A -85,B 0,C 180,E1 -961.056,E2 -961.056} C_VEL
LIN {X 0,Y 594.293,Z 173.336,A -85,B 0,C 180,E1 -963.295,E2 -963.295} C_VEL
LIN {X 0,Y 594.304,Z 176.508,A -85,B 0,C 180,E1 -965.585,E2 -965.585} C_VEL
LIN {X 0,Y 594.251,Z 179.49,A -85,B 0,C 180,E1 -967.761,E2 -967.761} C_VEL
LIN {X 0,Y 594.222,Z 182.763,A -85,B 0,C 180,E1 -969.94,E2 -969.94} C_VEL
LIN {X 0,Y 594.213,Z 186.067,A -85,B 0,C 180,E1 -972.09,E2 -972.09} C_VEL
LIN {X 0,Y 594.234,Z 189.371,A -85,B 0,C 180,E1 -974.215,E2 -974.215} C_VEL
LIN {X 0,Y 594.227,Z 193.777,A -85,B 0,C 180,E1 -977.013,E2 -977.013} C_VEL
LIN {X 0,Y 594.203,Z 198.183,A -85,B 0,C 180,E1 -979.78,E2 -979.78} C_VEL
LIN {X 0,Y 594.198,Z 202.589,A -85,B 0,C 180,E1 -982.524,E2 -982.524} C_VEL
LIN {X 0,Y 594.243,Z 203.449,A -85,B 0,C 180,E1 -983.058,E2 -983.058} C_VEL
LIN {X 0,Y 594.325,Z 212.866,A -85,B 0,C 180,E1 -983.413,E2 -983.413} C_VEL
LIN {X 0,Y 594.29,Z 221.954,A -85,B 0,C 180,E1 -983.889,E2 -983.889} C_VEL
LIN {X 0,Y 594.247,Z 230.291,A -85,B 0,C 180,E1 -984.485,E2 -984.485} C_VEL
LIN {X 0,Y 594.332,Z 236.746,A -85,B 0,C 180,E1 -985.081,E2 -985.081} C_VEL
LIN {X 0,Y 594.267,Z 242.56,A -85,B 0,C 180,E1 -985.76,E2 -985.76} C_VEL
LIN {X 0,Y 594.273,Z 248.026,A -85,B 0,C 180,E1 -986.609,E2 -986.609} C_VEL
LIN {X 0,Y 594.236,Z 251.35,A -85,B 0,C 180,E1 -987.288,E2 -987.288} C_VEL
LIN {X 0,Y 594.244,Z 253.836,A -85,B 0,C 180,E1 -987.966,E2 -987.966} C_VEL
LIN {X 0,Y 594.248,Z 255.566,A -85,B 0,C 180,E1 -988.644,E2 -988.644} C_VEL
LIN {X 0,Y 594.24,Z 256.599,A -85,B 0,C 180,E1 -989.321,E2 -989.321} C_VEL
LIN {X 0,Y 594.236,Z 256.978,A -85,B 0,C 180,E1 -989.999,E2 -989.999} C_VEL
LIN {X 0,Y 594.239,Z 256.706,A -85,B 0,C 180,E1 -990.677,E2 -990.677} C_VEL
LIN {X 0,Y 594.249,Z 255.767,A -85,B 0,C 180,E1 -991.354,E2 -991.354} C_VEL
LIN {X 0,Y 594.242,Z 254.13,A -85,B 0,C 180,E1 -992.032,E2 -992.032} C_VEL
LIN {X 0,Y 594.279,Z 250.245,A -85,B 0,C 180,E1 -993.05,E2 -993.05} C_VEL
LIN {X 0,Y 594.301,Z 245.54,A -85,B 0,C 180,E1 -993.898,E2 -993.898} C_VEL
LIN {X 0,Y 594.31,Z 240.555,A -85,B 0,C 180,E1 -994.577,E2 -994.577} C_VEL
LIN {X 0,Y 594.281,Z 234.247,A -85,B 0,C 180,E1 -995.258,E2 -995.258} C_VEL
LIN {X 0,Y 594.261,Z 227.08,A -85,B 0,C 180,E1 -995.854,E2 -995.854} C_VEL
LIN {X 0,Y 594.278,Z 219.129,A -85,B 0,C 180,E1 -996.363,E2 -996.363} C_VEL
LIN {X 0,Y 594.366,Z 210.226,A -85,B 0,C 180,E1 -996.79,E2 -996.79} C_VEL
LIN {X 0,Y 594.231,Z 203.425,A -85,B 0,C 180,E1 -997.047,E2 -997.047} C_VEL
LIN {X 0,Y 594.212,Z 199.431,A -85,B 0,C 180,E1 -999.53,E2 -999.53} C_VEL
LIN {X 0,Y 594.205,Z 196.126,A -85,B 0,C 180,E1 -1001.598,E2 -1001.598} C_VEL
LIN {X 0,Y 594.231,Z 191.719,A -85,B 0,C 180,E1 -1004.38,E2 -1004.38} C_VEL
LIN {X 0,Y 594.225,Z 187.311,A -85,B 0,C 180,E1 -1007.197,E2 -1007.197} C_VEL
LIN {X 0,Y 594.228,Z 184.005,A -85,B 0,C 180,E1 -1009.338,E2 -1009.338} C_VEL
LIN {X 0,Y 594.212,Z 180.7,A -85,B 0,C 180,E1 -1011.508,E2 -1011.508} C_VEL
LIN {X 0,Y 594.258,Z 177.619,A -85,B 0,C 180,E1 -1013.708,E2 -1013.708} C_VEL
LIN {X 0,Y 594.328,Z 174.431,A -85,B 0,C 180,E1 -1016.011,E2 -1016.011} C_VEL
LIN {X 0,Y 594.316,Z 171.359,A -85,B 0,C 180,E1 -1018.229,E2 -1018.229} C_VEL
LIN {X 0,Y 594.325,Z 169.458,A -85,B 0,C 180,E1 -1019.778,E2 -1019.778} C_VEL
LIN {X 0,Y 594.355,Z 169.447,A -85,B 0,C 180,E1 -1022.146,E2 -1022.146} C_VEL
LIN {X 0,Y 594.368,Z 169.443,A -85,B 0,C 180,E1 -1024.579,E2 -1024.579} C_VEL
LIN {X 0,Y 594.383,Z 169.447,A -85,B 0,C 180,E1 -1027.607,E2 -1027.607} C_VEL
LIN {X 0,Y 594.36,Z 169.445,A -85,B 0,C 180,E1 -1030.566,E2 -1030.566} C_VEL
LIN {X 0,Y 594.373,Z 169.449,A -85,B 0,C 180,E1 -1033.297,E2 -1033.297} C_VEL
LIN {X 0,Y 594.361,Z 169.444,A -85,B 0,C 180,E1 -1036.159,E2 -1036.159} C_VEL
LIN {X 0,Y 594.375,Z 169.446,A -85,B 0,C 180,E1 -1038.535,E2 -1038.535} C_VEL
LIN {X 0,Y 594.381,Z 169.443,A -85,B 0,C 180,E1 -1041.294,E2 -1041.294} C_VEL
LIN {X 0,Y 594.388,Z 169.44,A -85,B 0,C 180,E1 -1043.758,E2 -1043.758} C_VEL
LIN {X 0,Y 594.378,Z 169.447,A -85,B 0,C 180,E1 -1046.239,E2 -1046.239} C_VEL
LIN {X 0,Y 594.383,Z 169.446,A -85,B 0,C 180,E1 -1048.65,E2 -1048.65} C_VEL
LIN {X 0,Y 594.38,Z 169.442,A -85,B 0,C 180,E1 -1051.04,E2 -1051.04} C_VEL
LIN {X 0,Y 594.385,Z 169.447,A -85,B 0,C 180,E1 -1053.975,E2 -1053.975} C_VEL
LIN {X 0,Y 594.387,Z 169.446,A -85,B 0,C 180,E1 -1056.296,E2 -1056.296} C_VEL
LIN {X 0,Y 594.4,Z 169.439,A -85,B 0,C 180,E1 -1059.224,E2 -1059.224} C_VEL
LIN {X 0,Y 594.369,Z 169.447,A -85,B 0,C 180,E1 -1062.095,E2 -1062.095} C_VEL
LIN {X 0,Y 594.362,Z 169.445,A -85,B 0,C 180,E1 -1064.219,E2 -1064.219} C_VEL
LIN {X 0,Y 594.366,Z 169.445,A -85,B 0,C 180,E1 -1067.017,E2 -1067.017} C_VEL
LIN {X 0,Y 594.381,Z 169.445,A -85,B 0,C 180,E1 -1069.784,E2 -1069.784} C_VEL
LIN {X 0,Y 594.392,Z 169.44,A -85,B 0,C 180,E1 -1072.527,E2 -1072.527} C_VEL
LIN {X 0,Y 594.385,Z 169.449,A -85,B 0,C 180,E1 -1075.252,E2 -1075.252} C_VEL
LIN {X 0,Y 594.371,Z 169.442,A -85,B 0,C 180,E1 -1077.967,E2 -1077.967} C_VEL
LIN {X 0,Y 594.423,Z 169.441,A -85,B 0,C 180,E1 -1080.677,E2 -1080.677} C_VEL
LIN {X 0,Y 594.353,Z 169.446,A -85,B 0,C 180,E1 -1083.389,E2 -1083.389} C_VEL
LIN {X 0,Y 594.363,Z 169.444,A -85,B 0,C 180,E1 -1085.428,E2 -1085.428} C_VEL
LIN {X 0,Y 594.399,Z 169.442,A -85,B 0,C 180,E1 -1088.157,E2 -1088.157} C_VEL
LIN {X 0,Y 594.365,Z 169.445,A -85,B 0,C 180,E1 -1091.068,E2 -1091.068} C_VEL
LIN {X 0,Y 594.355,Z 169.445,A -85,B 0,C 180,E1 -1093.68,E2 -1093.68} C_VEL
LIN {X 0,Y 594.368,Z 169.448,A -85,B 0,C 180,E1 -1096.486,E2 -1096.486} C_VEL
LIN {X 0,Y 594.343,Z 169.446,A -85,B 0,C 180,E1 -1099.335,E2 -1099.335} C_VEL
LIN {X 0,Y 594.334,Z 169.45,A -85,B 0,C 180,E1 -1101.505,E2 -1101.505} C_VEL
LIN {X 0,Y 594.353,Z 169.446,A -85,B 0,C 180,E1 -1104.448,E2 -1104.448} C_VEL
LIN {X 0,Y 594.331,Z 169.447,A -85,B 0,C 180,E1 -1106.702,E2 -1106.702} C_VEL
LIN {X 0,Y 594.344,Z 169.453,A -85,B 0,C 180,E1 -1109.778,E2 -1109.778} C_VEL
LIN {X 0,Y 594.331,Z 169.449,A -85,B 0,C 180,E1 -1112.149,E2 -1112.149} C_VEL
LIN {X 0,Y 594.353,Z 169.445,A -85,B 0,C 180,E1 -1114.582,E2 -1114.582} C_VEL
LIN {X 0,Y 594.374,Z 169.447,A -85,B 0,C 180,E1 -1117.609,E2 -1117.609} C_VEL
LIN {X 0,Y 594.352,Z 169.446,A -85,B 0,C 180,E1 -1120.569,E2 -1120.569} C_VEL
LIN {X 0,Y 594.353,Z 169.449,A -85,B 0,C 180,E1 -1123.301,E2 -1123.301} C_VEL
LIN {X 0,Y 594.352,Z 169.446,A -85,B 0,C 180,E1 -1126.162,E2 -1126.162} C_VEL
LIN {X 0,Y 594.369,Z 169.446,A -85,B 0,C 180,E1 -1129.179,E2 -1129.179} C_VEL
LIN {X 0,Y 594.369,Z 169.445,A -85,B 0,C 180,E1 -1132.06,E2 -1132.06} C_VEL
LIN {X 0,Y 594.354,Z 169.451,A -85,B 0,C 180,E1 -1134.677,E2 -1134.677} C_VEL
LIN {X 0,Y 594.371,Z 169.444,A -85,B 0,C 180,E1 -1137.09,E2 -1137.09} C_VEL
LIN {X 0,Y 594.367,Z 169.447,A -85,B 0,C 180,E1 -1139.676,E2 -1139.676} C_VEL
LIN {X 0,Y 594.42,Z 169.597,A -85,B 0,C 180,E1 -1140.714,E2 -1140.714} C_VEL
LIN {X 0,Y 595.103,Z 174.109,A -85,B 0,C 180,E1 -1141.427,E2 -1141.427} C_VEL
LIN {X 0,Y 594.975,Z 191.125,A -85,B 0,C 180,E1 -1143.862,E2 -1143.862} C_VEL
LIN {X 0,Y 594.83,Z 211.317,A -85,B 0,C 180,E1 -1146.685,E2 -1146.685} C_VEL
LIN {X 0,Y 594.695,Z 229.931,A -85,B 0,C 180,E1 -1149.236,E2 -1149.236} C_VEL
LIN {X 0,Y 594.603,Z 251.205,A -85,B 0,C 180,E1 -1152.104,E2 -1152.104} C_VEL
LIN {X 0,Y 594.474,Z 272.478,A -85,B 0,C 180,E1 -1154.926,E2 -1154.926} C_VEL
LIN {X 0,Y 594.4,Z 292.422,A -85,B 0,C 180,E1 -1157.54,E2 -1157.54} C_VEL
LIN {X 0,Y 594.406,Z 294.915,A -85,B 0,C 180,E1 -1157.865,E2 -1157.865} C_VEL
LIN {X 0,Y 594.688,Z 298.669,A -85,B 0,C 180,E1 -1157.935,E2 -1157.935} C_VEL
LIN {X 0,Y 594.626,Z 312.221,A -85,B 0,C 180,E1 -1158.194,E2 -1158.194} C_VEL
LIN {X 0,Y 594.574,Z 324.874,A -85,B 0,C 180,E1 -1158.576,E2 -1158.576} C_VEL
LIN {X 0,Y 594.554,Z 337.197,A -85,B 0,C 180,E1 -1159.099,E2 -1159.099} C_VEL
LIN {X 0,Y 594.462,Z 349.598,A -85,B 0,C 180,E1 -1159.786,E2 -1159.786} C_VEL
LIN {X 0,Y 594.422,Z 360.488,A -85,B 0,C 180,E1 -1160.559,E2 -1160.559} C_VEL
LIN {X 0,Y 594.383,Z 371.122,A -85,B 0,C 180,E1 -1161.501,E2 -1161.501} C_VEL
LIN {X 0,Y 594.347,Z 378.968,A -85,B 0,C 180,E1 -1162.356,E2 -1162.356} C_VEL
LIN {X 0,Y 594.282,Z 386.817,A -85,B 0,C 180,E1 -1163.409,E2 -1163.409} C_VEL
LIN {X 0,Y 594.289,Z 393.685,A -85,B 0,C 180,E1 -1164.572,E2 -1164.572} C_VEL
LIN {X 0,Y 594.27,Z 398.375,A -85,B 0,C 180,E1 -1165.592,E2 -1165.592} C_VEL
LIN {X 0,Y 594.267,Z 401.96,A -85,B 0,C 180,E1 -1166.611,E2 -1166.611} C_VEL
LIN {X 0,Y 594.226,Z 403.812,A -85,B 0,C 180,E1 -1167.289,E2 -1167.289} C_VEL
LIN {X 0,Y 594.242,Z 405.203,A -85,B 0,C 180,E1 -1167.968,E2 -1167.968} C_VEL
LIN {X 0,Y 594.239,Z 406.785,A -85,B 0,C 180,E1 -1169.323,E2 -1169.323} C_VEL
LIN {X 0,Y 594.236,Z 407,A -85,B 0,C 180,E1 -1170.001,E2 -1170.001} C_VEL
LIN {X 0,Y 594.247,Z 406.184,A -85,B 0,C 180,E1 -1171.356,E2 -1171.356} C_VEL
LIN {X 0,Y 594.242,Z 405.2,A -85,B 0,C 180,E1 -1172.034,E2 -1172.034} C_VEL
LIN {X 0,Y 594.226,Z 403.807,A -85,B 0,C 180,E1 -1172.712,E2 -1172.712} C_VEL
LIN {X 0,Y 594.289,Z 400.893,A -85,B 0,C 180,E1 -1173.73,E2 -1173.73} C_VEL
LIN {X 0,Y 594.241,Z 396.946,A -85,B 0,C 180,E1 -1174.75,E2 -1174.75} C_VEL
LIN {X 0,Y 594.305,Z 390.872,A -85,B 0,C 180,E1 -1175.94,E2 -1175.94} C_VEL
LIN {X 0,Y 594.309,Z 384.23,A -85,B 0,C 180,E1 -1176.963,E2 -1176.963} C_VEL
LIN {X 0,Y 594.36,Z 375.983,A -85,B 0,C 180,E1 -1177.987,E2 -1177.987} C_VEL
LIN {X 0,Y 594.382,Z 367.528,A -85,B 0,C 180,E1 -1178.843,E2 -1178.843} C_VEL
LIN {X 0,Y 594.431,Z 357.083,A -85,B 0,C 180,E1 -1179.7,E2 -1179.7} C_VEL
LIN {X 0,Y 594.477,Z 346.745,A -85,B 0,C 180,E1 -1180.387,E2 -1180.387} C_VEL
LIN {X 0,Y 594.557,Z 335.732,A -85,B 0,C 180,E1 -1180.973,E2 -1180.973} C_VEL
LIN {X 0,Y 594.581,Z 323.698,A -85,B 0,C 180,E1 -1181.465,E2 -1181.465} C_VEL
LIN {X 0,Y 594.636,Z 310.321,A -85,B 0,C 180,E1 -1181.851,E2 -1181.851} C_VEL
LIN {X 0,Y 594.664,Z 297.025,A -85,B 0,C 180,E1 -1182.088,E2 -1182.088} C_VEL
LIN {X 0,Y 594.407,Z 294.902,A -85,B 0,C 180,E1 -1182.137,E2 -1182.137} C_VEL
LIN {X 0,Y 594.459,Z 273.794,A -85,B 0,C 180,E1 -1184.901,E2 -1184.901} C_VEL
LIN {X 0,Y 594.577,Z 253.85,A -85,B 0,C 180,E1 -1187.543,E2 -1187.543} C_VEL
LIN {X 0,Y 594.696,Z 232.577,A -85,B 0,C 180,E1 -1190.404,E2 -1190.404} C_VEL
LIN {X 0,Y 594.84,Z 212.633,A -85,B 0,C 180,E1 -1193.132,E2 -1193.132} C_VEL
LIN {X 0,Y 594.968,Z 191.137,A -85,B 0,C 180,E1 -1196.137,E2 -1196.137} C_VEL
LIN {X 0,Y 595.139,Z 174.191,A -85,B 0,C 180,E1 -1198.573,E2 -1198.573} C_VEL
LIN {X 0,Y 594.38,Z 169.45,A -85,B 0,C 180,E1 -1199.338,E2 -1199.338} C_VEL
LIN {X 0,Y 594.344,Z 169.449,A -85,B 0,C 180,E1 -1202.149,E2 -1202.149} C_VEL
LIN {X 0,Y 594.366,Z 169.448,A -85,B 0,C 180,E1 -1204.582,E2 -1204.582} C_VEL
LIN {X 0,Y 594.386,Z 169.442,A -85,B 0,C 180,E1 -1207.608,E2 -1207.608} C_VEL
LIN {X 0,Y 594.369,Z 169.448,A -85,B 0,C 180,E1 -1210.568,E2 -1210.568} C_VEL
LIN {X 0,Y 594.37,Z 169.445,A -85,B 0,C 180,E1 -1213.3,E2 -1213.3} C_VEL
LIN {X 0,Y 594.365,Z 169.446,A -85,B 0,C 180,E1 -1216.162,E2 -1216.162} C_VEL
LIN {X 0,Y 594.381,Z 169.444,A -85,B 0,C 180,E1 -1218.536,E2 -1218.536} C_VEL
LIN {X 0,Y 594.367,Z 169.448,A -85,B 0,C 180,E1 -1221.298,E2 -1221.298} C_VEL
LIN {X 0,Y 594.339,Z 169.449,A -85,B 0,C 180,E1 -1223.754,E2 -1223.754} C_VEL
LIN {X 0,Y 594.314,Z 169.565,A -85,B 0,C 180,E1 -1226.022,E2 -1226.022} C_VEL
LIN {X 0,Y 594.324,Z 178.291,A -85,B 0,C 180,E1 -1228.367,E2 -1228.367} C_VEL
LIN {X 0,Y 594.347,Z 187.604,A -85,B 0,C 180,E1 -1231.049,E2 -1231.049} C_VEL
LIN {X 0,Y 594.39,Z 196.028,A -85,B 0,C 180,E1 -1233.675,E2 -1233.675} C_VEL
LIN {X 0,Y 594.393,Z 203.973,A -85,B 0,C 180,E1 -1236.296,E2 -1236.296} C_VEL
LIN {X 0,Y 594.353,Z 212.875,A -85,B 0,C 180,E1 -1239.223,E2 -1239.223} C_VEL
LIN {X 0,Y 594.332,Z 221.777,A -85,B 0,C 180,E1 -1242.094,E2 -1242.094} C_VEL
LIN {X 0,Y 594.292,Z 230.679,A -85,B 0,C 180,E1 -1244.92,E2 -1244.92} C_VEL
LIN {X 0,Y 594.293,Z 239.582,A -85,B 0,C 180,E1 -1247.71,E2 -1247.71} C_VEL
LIN {X 0,Y 594.302,Z 240.728,A -85,B 0,C 180,E1 -1248.002,E2 -1248.002} C_VEL
LIN {X 0,Y 594.676,Z 246.32,A -85,B 0,C 180,E1 -1248.107,E2 -1248.107} C_VEL
LIN {X 0,Y 594.594,Z 259.838,A -85,B 0,C 180,E1 -1248.451,E2 -1248.451} C_VEL
LIN {X 0,Y 594.537,Z 272.265,A -85,B 0,C 180,E1 -1248.917,E2 -1248.917} C_VEL
LIN {X 0,Y 594.506,Z 284.521,A -85,B 0,C 180,E1 -1249.528,E2 -1249.528} C_VEL
LIN {X 0,Y 594.449,Z 295.319,A -85,B 0,C 180,E1 -1250.215,E2 -1250.215} C_VEL
LIN {X 0,Y 594.404,Z 305.093,A -85,B 0,C 180,E1 -1250.987,E2 -1250.987} C_VEL
LIN {X 0,Y 594.366,Z 313.99,A -85,B 0,C 180,E1 -1251.843,E2 -1251.843} C_VEL
LIN {X 0,Y 594.308,Z 322.664,A -85,B 0,C 180,E1 -1252.867,E2 -1252.867} C_VEL
LIN {X 0,Y 594.29,Z 329.605,A -85,B 0,C 180,E1 -1253.89,E2 -1253.89} C_VEL
LIN {X 0,Y 594.254,Z 335.158,A -85,B 0,C 180,E1 -1254.911,E2 -1254.911} C_VEL
LIN {X 0,Y 594.263,Z 339.518,A -85,B 0,C 180,E1 -1255.931,E2 -1255.931} C_VEL
LIN {X 0,Y 594.267,Z 341.82,A -85,B 0,C 180,E1 -1256.61,E2 -1256.61} C_VEL
LIN {X 0,Y 594.225,Z 343.692,A -85,B 0,C 180,E1 -1257.288,E2 -1257.288} C_VEL
LIN {X 0,Y 594.24,Z 345.13,A -85,B 0,C 180,E1 -1257.967,E2 -1257.967} C_VEL
LIN {X 0,Y 594.241,Z 346.753,A -85,B 0,C 180,E1 -1259.322,E2 -1259.322} C_VEL
LIN {X 0,Y 594.236,Z 346.996,A -85,B 0,C 180,E1 -1260,E2 -1260} C_VEL
LIN {X 0,Y 594.239,Z 346.814,A -85,B 0,C 180,E1 -1260.678,E2 -1260.678} C_VEL
LIN {X 0,Y 594.239,Z 345.276,A -85,B 0,C 180,E1 -1262.033,E2 -1262.033} C_VEL
LIN {X 0,Y 594.226,Z 343.915,A -85,B 0,C 180,E1 -1262.712,E2 -1262.712} C_VEL
LIN {X 0,Y 594.289,Z 341.043,A -85,B 0,C 180,E1 -1263.729,E2 -1263.729} C_VEL
LIN {X 0,Y 594.242,Z 337.144,A -85,B 0,C 180,E1 -1264.749,E2 -1264.749} C_VEL
LIN {X 0,Y 594.299,Z 332.112,A -85,B 0,C 180,E1 -1265.769,E2 -1265.769} C_VEL
LIN {X 0,Y 594.317,Z 325.781,A -85,B 0,C 180,E1 -1266.791,E2 -1266.791} C_VEL
LIN {X 0,Y 594.347,Z 317.874,A -85,B 0,C 180,E1 -1267.816,E2 -1267.816} C_VEL
LIN {X 0,Y 594.377,Z 309.805,A -85,B 0,C 180,E1 -1268.671,E2 -1268.671} C_VEL
LIN {X 0,Y 594.417,Z 299.964,A -85,B 0,C 180,E1 -1269.528,E2 -1269.528} C_VEL
LIN {X 0,Y 594.431,Z 288.906,A -85,B 0,C 180,E1 -1270.301,E2 -1270.301} C_VEL
LIN {X 0,Y 594.5,Z 278.087,A -85,B 0,C 180,E1 -1270.903,E2 -1270.903} C_VEL
LIN {X 0,Y 594.578,Z 266.251,A -85,B 0,C 180,E1 -1271.416,E2 -1271.416} C_VEL
LIN {X 0,Y 594.637,Z 253.728,A -85,B 0,C 180,E1 -1271.814,E2 -1271.814} C_VEL
LIN {X 0,Y 593.94,Z 249.792,A -85,B 0,C 180,E1 -1271.936,E2 -1271.936} C_VEL
LIN {X 0,Y 591.6,Z 245.157,A -85,B 0,C 180,E1 -1272.159,E2 -1272.159} C_VEL
LIN {X 0,Y 588.971,Z 241.353,A -85,B 0,C 180,E1 -1272.464,E2 -1272.464} C_VEL
LIN {X 0,Y 587.453,Z 238.966,A -85,B 0,C 180,E1 -1272.797,E2 -1272.797} C_VEL
LIN {X 0,Y 587.193,Z 238.073,A -85,B 0,C 180,E1 -1273.008,E2 -1273.008} C_VEL
LIN {X 0,Y 587.209,Z 228.736,A -85,B 0,C 180,E1 -1275.979,E2 -1275.979} C_VEL
LIN {X 0,Y 587.248,Z 219.829,A -85,B 0,C 180,E1 -1278.852,E2 -1278.852} C_VEL
LIN {X 0,Y 587.284,Z 212.036,A -85,B 0,C 180,E1 -1281.407,E2 -1281.407} C_VEL
LIN {X 0,Y 587.289,Z 204.242,A -85,B 0,C 180,E1 -1284.009,E2 -1284.009} C_VEL
LIN {X 0,Y 587.353,Z 196.396,A -85,B 0,C 180,E1 -1286.661,E2 -1286.661} C_VEL
LIN {X 0,Y 587.367,Z 188.151,A -85,B 0,C 180,E1 -1289.379,E2 -1289.379} C_VEL
LIN {X 0,Y 587.418,Z 179.656,A -85,B 0,C 180,E1 -1292.173,E2 -1292.173} C_VEL
LIN {X 0,Y 587.394,Z 170.917,A -85,B 0,C 180,E1 -1295.051,E2 -1295.051} C_VEL
LIN {X 0,Y 587.312,Z 170.328,A -85,B 0,C 180,E1 -1295.315,E2 -1295.315} C_VEL
LIN {X 0,Y 587.329,Z 170.329,A -85,B 0,C 180,E1 -1297.836,E2 -1297.836} C_VEL
LIN {X 0,Y 587.315,Z 170.324,A -85,B 0,C 180,E1 -1300.255,E2 -1300.255} C_VEL
LIN {X 0,Y 587.306,Z 170.327,A -85,B 0,C 180,E1 -1303.117,E2 -1303.117} C_VEL
LIN {X 0,Y 587.318,Z 170.329,A -85,B 0,C 180,E1 -1306.048,E2 -1306.048} C_VEL
LIN {X 0,Y 587.339,Z 170.325,A -85,B 0,C 180,E1 -1308.925,E2 -1308.925} C_VEL
LIN {X 0,Y 587.321,Z 170.324,A -85,B 0,C 180,E1 -1311.519,E2 -1311.519} C_VEL
LIN {X 0,Y 587.28,Z 170.334,A -85,B 0,C 180,E1 -1314.098,E2 -1314.098} C_VEL
LIN {X 0,Y 587.341,Z 170.325,A -85,B 0,C 180,E1 -1316.889,E2 -1316.889} C_VEL
LIN {X 0,Y 587.342,Z 170.321,A -85,B 0,C 180,E1 -1319.49,E2 -1319.49} C_VEL
LIN {X 0,Y 587.246,Z 170.385,A -85,B 0,C 180,E1 -1320.614,E2 -1320.614} C_VEL
LIN {X 0,Y 587.237,Z 173.587,A -85,B 0,C 180,E1 -1322.948,E2 -1322.948} C_VEL
LIN {X 0,Y 587.219,Z 177.044,A -85,B 0,C 180,E1 -1325.449,E2 -1325.449} C_VEL
LIN {X 0,Y 587.144,Z 180.773,A -85,B 0,C 180,E1 -1328.218,E2 -1328.218} C_VEL
LIN {X 0,Y 587.129,Z 183.865,A -85,B 0,C 180,E1 -1330.417,E2 -1330.417} C_VEL
LIN {X 0,Y 587.17,Z 188.271,A -85,B 0,C 180,E1 -1333.305,E2 -1333.305} C_VEL
LIN {X 0,Y 587.165,Z 192.676,A -85,B 0,C 180,E1 -1336.149,E2 -1336.149} C_VEL
LIN {X 0,Y 587.168,Z 197.082,A -85,B 0,C 180,E1 -1338.958,E2 -1338.958} C_VEL
LIN {X 0,Y 587.112,Z 201.488,A -85,B 0,C 180,E1 -1341.74,E2 -1341.74} C_VEL
LIN {X 0,Y 587.133,Z 203.45,A -85,B 0,C 180,E1 -1342.973,E2 -1342.973} C_VEL
LIN {X 0,Y 587.293,Z 212.188,A -85,B 0,C 180,E1 -1343.304,E2 -1343.304} C_VEL
LIN {X 0,Y 587.251,Z 220.086,A -85,B 0,C 180,E1 -1343.707,E2 -1343.707} C_VEL
LIN {X 0,Y 587.194,Z 228.153,A -85,B 0,C 180,E1 -1344.246,E2 -1344.246} C_VEL
LIN {X 0,Y 587.257,Z 235.06,A -85,B 0,C 180,E1 -1344.85,E2 -1344.85} C_VEL
LIN {X 0,Y 587.216,Z 241.214,A -85,B 0,C 180,E1 -1345.537,E2 -1345.537} C_VEL
LIN {X 0,Y 587.228,Z 246.061,A -85,B 0,C 180,E1 -1346.225,E2 -1346.225} C_VEL
LIN {X 0,Y 587.184,Z 249.821,A -85,B 0,C 180,E1 -1346.912,E2 -1346.912} C_VEL
LIN {X 0,Y 587.145,Z 253.843,A -85,B 0,C 180,E1 -1347.941,E2 -1347.941} C_VEL
LIN {X 0,Y 587.147,Z 255.566,A -85,B 0,C 180,E1 -1348.627,E2 -1348.627} C_VEL
LIN {X 0,Y 587.14,Z 256.591,A -85,B 0,C 180,E1 -1349.313,E2 -1349.313} C_VEL
LIN {X 0,Y 587.137,Z 256.968,A -85,B 0,C 180,E1 -1349.999,E2 -1349.999} C_VEL
LIN {X 0,Y 587.14,Z 256.7,A -85,B 0,C 180,E1 -1350.685,E2 -1350.685} C_VEL
LIN {X 0,Y 587.148,Z 255.766,A -85,B 0,C 180,E1 -1351.371,E2 -1351.371} C_VEL
LIN {X 0,Y 587.172,Z 253.004,A -85,B 0,C 180,E1 -1352.4,E2 -1352.4} C_VEL
LIN {X 0,Y 587.184,Z 250.25,A -85,B 0,C 180,E1 -1353.087,E2 -1353.087} C_VEL
LIN {X 0,Y 587.223,Z 245.529,A -85,B 0,C 180,E1 -1353.945,E2 -1353.945} C_VEL
LIN {X 0,Y 587.241,Z 240.551,A -85,B 0,C 180,E1 -1354.633,E2 -1354.633} C_VEL
LIN {X 0,Y 587.205,Z 234.228,A -85,B 0,C 180,E1 -1355.321,E2 -1355.321} C_VEL
LIN {X 0,Y 587.198,Z 227.059,A -85,B 0,C 180,E1 -1355.924,E2 -1355.924} C_VEL
LIN {X 0,Y 587.228,Z 219.109,A -85,B 0,C 180,E1 -1356.439,E2 -1356.439} C_VEL
LIN {X 0,Y 587.332,Z 210.191,A -85,B 0,C 180,E1 -1356.872,E2 -1356.872} C_VEL
LIN {X 0,Y 587.141,Z 203.424,A -85,B 0,C 180,E1 -1357.133,E2 -1357.133} C_VEL
LIN {X 0,Y 587.111,Z 199.43,A -85,B 0,C 180,E1 -1359.647,E2 -1359.647} C_VEL
LIN {X 0,Y 587.131,Z 196.125,A -85,B 0,C 180,E1 -1361.74,E2 -1361.74} C_VEL
LIN {X 0,Y 587.123,Z 191.718,A -85,B 0,C 180,E1 -1364.558,E2 -1364.558} C_VEL
LIN {X 0,Y 587.144,Z 188.331,A -85,B 0,C 180,E1 -1366.746,E2 -1366.746} C_VEL
LIN {X 0,Y 587.125,Z 184.005,A -85,B 0,C 180,E1 -1369.581,E2 -1369.581} C_VEL
LIN {X 0,Y 587.14,Z 180.907,A -85,B 0,C 180,E1 -1371.78,E2 -1371.78} C_VEL
LIN {X 0,Y 587.213,Z 177.135,A -85,B 0,C 180,E1 -1374.549,E2 -1374.549} C_VEL
LIN {X 0,Y 587.236,Z 173.742,A -85,B 0,C 180,E1 -1377.05,E2 -1377.05} C_VEL
LIN {X 0,Y 587.247,Z 170.507,A -85,B 0,C 180,E1 -1379.384,E2 -1379.384} C_VEL
LIN {X 0,Y 587.334,Z 170.327,A -85,B 0,C 180,E1 -1381.768,E2 -1381.768} C_VEL
LIN {X 0,Y 587.341,Z 170.319,A -85,B 0,C 180,E1 -1384.346,E2 -1384.346} C_VEL
LIN {X 0,Y 587.345,Z 170.319,A -85,B 0,C 180,E1 -1386.746,E2 -1386.746} C_VEL
LIN {X 0,Y 587.338,Z 170.327,A -85,B 0,C 180,E1 -1389.358,E2 -1389.358} C_VEL
LIN {X 0,Y 587.329,Z 170.32,A -85,B 0,C 180,E1 -1392.107,E2 -1392.107} C_VEL
LIN {X 0,Y 587.311,Z 170.331,A -85,B 0,C 180,E1 -1395.088,E2 -1395.088} C_VEL
LIN {X 0,Y 587.346,Z 170.318,A -85,B 0,C 180,E1 -1397.927,E2 -1397.927} C_VEL
LIN {X 0,Y 587.328,Z 170.325,A -85,B 0,C 180,E1 -1401.057,E2 -1401.057} C_VEL
LIN {X 0,Y 587.347,Z 170.319,A -85,B 0,C 180,E1 -1403.291,E2 -1403.291} C_VEL
LIN {X 0,Y 587.363,Z 170.316,A -85,B 0,C 180,E1 -1405.78,E2 -1405.78} C_VEL
LIN {X 0,Y 587.347,Z 170.324,A -85,B 0,C 180,E1 -1408.231,E2 -1408.231} C_VEL
LIN {X 0,Y 587.346,Z 170.319,A -85,B 0,C 180,E1 -1410.865,E2 -1410.865} C_VEL
LIN {X 0,Y 587.354,Z 170.321,A -85,B 0,C 180,E1 -1413.817,E2 -1413.817} C_VEL
LIN {X 0,Y 587.316,Z 170.322,A -85,B 0,C 180,E1 -1416.741,E2 -1416.741} C_VEL
LIN {X 0,Y 587.326,Z 170.326,A -85,B 0,C 180,E1 -1419.695,E2 -1419.695} C_VEL
LIN {X 0,Y 587.347,Z 170.318,A -85,B 0,C 180,E1 -1422.594,E2 -1422.594} C_VEL
LIN {X 0,Y 587.354,Z 170.324,A -85,B 0,C 180,E1 -1425.739,E2 -1425.739} C_VEL
LIN {X 0,Y 587.351,Z 170.318,A -85,B 0,C 180,E1 -1428.858,E2 -1428.858} C_VEL
LIN {X 0,Y 587.359,Z 170.319,A -85,B 0,C 180,E1 -1431.745,E2 -1431.745} C_VEL
LIN {X 0,Y 587.353,Z 170.317,A -85,B 0,C 180,E1 -1434.507,E2 -1434.507} C_VEL
LIN {X 0,Y 587.362,Z 170.322,A -85,B 0,C 180,E1 -1437.257,E2 -1437.257} C_VEL
LIN {X 0,Y 587.359,Z 170.315,A -85,B 0,C 180,E1 -1440,E2 -1440} C_VEL
LIN {X 0,Y 587.372,Z 170.322,A -85,B 0,C 180,E1 -1442.743,E2 -1442.743} C_VEL
LIN {X 0,Y 587.329,Z 170.32,A -85,B 0,C 180,E1 -1445.493,E2 -1445.493} C_VEL
LIN {X 0,Y 587.354,Z 170.321,A -85,B 0,C 180,E1 -1448.255,E2 -1448.255} C_VEL
LIN {X 0,Y 587.336,Z 170.32,A -85,B 0,C 180,E1 -1451.134,E2 -1451.134} C_VEL
LIN {X 0,Y 587.351,Z 170.325,A -85,B 0,C 180,E1 -1454.26,E2 -1454.26} C_VEL
LIN {X 0,Y 587.293,Z 170.324,A -85,B 0,C 180,E1 -1457.408,E2 -1457.408} C_VEL
LIN {X 0,Y 587.289,Z 170.327,A -85,B 0,C 180,E1 -1459.577,E2 -1459.577} C_VEL
LIN {X 0,Y 587.292,Z 170.331,A -85,B 0,C 180,E1 -1461.776,E2 -1461.776} C_VEL
LIN {X 0,Y 587.288,Z 170.325,A -85,B 0,C 180,E1 -1464.761,E2 -1464.761} C_VEL
LIN {X 0,Y 587.283,Z 170.335,A -85,B 0,C 180,E1 -1467.683,E2 -1467.683} C_VEL
LIN {X 0,Y 587.304,Z 170.323,A -85,B 0,C 180,E1 -1470.507,E2 -1470.507} C_VEL
LIN {X 0,Y 587.32,Z 170.33,A -85,B 0,C 180,E1 -1473.398,E2 -1473.398} C_VEL
LIN {X 0,Y 587.268,Z 170.329,A -85,B 0,C 180,E1 -1475.902,E2 -1475.902} C_VEL
LIN {X 0,Y 587.304,Z 170.324,A -85,B 0,C 180,E1 -1478.482,E2 -1478.482} C_VEL
LIN {X 0,Y 587.327,Z 170.329,A -85,B 0,C 180,E1 -1481.158,E2 -1481.158} C_VEL
LIN {X 0,Y 587.304,Z 170.323,A -85,B 0,C 180,E1 -1484.113,E2 -1484.113} C_VEL
LIN {X 0,Y 587.306,Z 170.329,A -85,B 0,C 180,E1 -1486.994,E2 -1486.994} C_VEL
LIN {X 0,Y 587.307,Z 170.323,A -85,B 0,C 180,E1 -1489.747,E2 -1489.747} C_VEL
LIN {X 0,Y 587.336,Z 170.326,A -85,B 0,C 180,E1 -1492.393,E2 -1492.393} C_VEL
LIN {X 0,Y 587.345,Z 170.319,A -85,B 0,C 180,E1 -1495.653,E2 -1495.653} C_VEL
LIN {X 0,Y 587.344,Z 170.327,A -85,B 0,C 180,E1 -1498.233,E2 -1498.233} C_VEL
LIN {X 0,Y 587.348,Z 170.409,A -85,B 0,C 180,E1 -1500.45,E2 -1500.45} C_VEL
LIN {X 0,Y 588.321,Z 175.598,A -85,B 0,C 180,E1 -1501.284,E2 -1501.284} C_VEL
LIN {X 0,Y 588.139,Z 192.636,A -85,B 0,C 180,E1 -1503.761,E2 -1503.761} C_VEL
LIN {X 0,Y 587.938,Z 212.647,A -85,B 0,C 180,E1 -1506.582,E2 -1506.582} C_VEL
LIN {X 0,Y 587.769,Z 231.261,A -85,B 0,C 180,E1 -1509.163,E2 -1509.163} C_VEL
LIN {X 0,Y 587.645,Z 251.205,A -85,B 0,C 180,E1 -1511.885,E2 -1511.885} C_VEL
LIN {X 0,Y 587.492,Z 272.478,A -85,B 0,C 180,E1 -1514.742,E2 -1514.742} C_VEL
LIN {X 0,Y 587.391,Z 292.422,A -85,B 0,C 180,E1 -1517.388,E2 -1517.388} C_VEL
LIN {X 0,Y 587.359,Z 294.915,A -85,B 0,C 180,E1 -1517.717,E2 -1517.717} C_VEL
LIN {X 0,Y 587.752,Z 298.669,A -85,B 0,C 180,E1 -1517.791,E2 -1517.791} C_VEL
LIN {X 0,Y 587.696,Z 312.22,A -85,B 0,C 180,E1 -1518.053,E2 -1518.053} C_VEL
LIN {X 0,Y 587.621,Z 324.721,A -85,B 0,C 180,E1 -1518.434,E2 -1518.434} C_VEL
LIN {X 0,Y 587.566,Z 337.199,A -85,B 0,C 180,E1 -1518.968,E2 -1518.968} C_VEL
LIN {X 0,Y 587.459,Z 349.6,A -85,B 0,C 180,E1 -1519.663,E2 -1519.663} C_VEL
LIN {X 0,Y 587.397,Z 360.486,A -85,B 0,C 180,E1 -1520.445,E2 -1520.445} C_VEL
LIN {X 0,Y 587.321,Z 371.122,A -85,B 0,C 180,E1 -1521.399,E2 -1521.399} C_VEL
LIN {X 0,Y 587.273,Z 378.968,A -85,B 0,C 180,E1 -1522.264,E2 -1522.264} C_VEL
LIN {X 0,Y 587.231,Z 385.476,A -85,B 0,C 180,E1 -1523.127,E2 -1523.127} C_VEL
LIN {X 0,Y 587.237,Z 391.871,A -85,B 0,C 180,E1 -1524.162,E2 -1524.162} C_VEL
LIN {X 0,Y 587.147,Z 396.953,A -85,B 0,C 180,E1 -1525.195,E2 -1525.195} C_VEL
LIN {X 0,Y 587.213,Z 400.899,A -85,B 0,C 180,E1 -1526.227,E2 -1526.227} C_VEL
LIN {X 0,Y 587.132,Z 403.812,A -85,B 0,C 180,E1 -1527.257,E2 -1527.257} C_VEL
LIN {X 0,Y 587.141,Z 405.202,A -85,B 0,C 180,E1 -1527.943,E2 -1527.943} C_VEL
LIN {X 0,Y 587.14,Z 406.785,A -85,B 0,C 180,E1 -1529.315,E2 -1529.315} C_VEL
LIN {X 0,Y 587.137,Z 407,A -85,B 0,C 180,E1 -1530.001,E2 -1530.001} C_VEL
LIN {X 0,Y 587.147,Z 406.184,A -85,B 0,C 180,E1 -1531.373,E2 -1531.373} C_VEL
LIN {X 0,Y 587.141,Z 405.199,A -85,B 0,C 180,E1 -1532.059,E2 -1532.059} C_VEL
LIN {X 0,Y 587.132,Z 403.807,A -85,B 0,C 180,E1 -1532.745,E2 -1532.745} C_VEL
LIN {X 0,Y 587.213,Z 400.893,A -85,B 0,C 180,E1 -1533.775,E2 -1533.775} C_VEL
LIN {X 0,Y 587.147,Z 396.946,A -85,B 0,C 180,E1 -1534.807,E2 -1534.807} C_VEL
LIN {X 0,Y 587.218,Z 390.872,A -85,B 0,C 180,E1 -1536.012,E2 -1536.012} C_VEL
LIN {X 0,Y 587.246,Z 384.231,A -85,B 0,C 180,E1 -1537.047,E2 -1537.047} C_VEL
LIN {X 0,Y 587.3,Z 375.983,A -85,B 0,C 180,E1 -1538.084,E2 -1538.084} C_VEL
LIN {X 0,Y 587.344,Z 367.529,A -85,B 0,C 180,E1 -1538.95,E2 -1538.95} C_VEL
LIN {X 0,Y 587.417,Z 357.085,A -85,B 0,C 180,E1 -1539.817,E2 -1539.817} C_VEL
LIN {X 0,Y 587.485,Z 346.744,A -85,B 0,C 180,E1 -1540.512,E2 -1540.512} C_VEL
LIN {X 0,Y 587.569,Z 334.969,A -85,B 0,C 180,E1 -1541.142,E2 -1541.142} C_VEL
LIN {X 0,Y 587.623,Z 322.581,A -85,B 0,C 180,E1 -1541.64,E2 -1541.64} C_VEL
LIN {X 0,Y 587.691,Z 309.405,A -85,B 0,C 180,E1 -1542.015,E2 -1542.015} C_VEL
LIN {X 0,Y 587.664,Z 297.026,A -85,B 0,C 180,E1 -1542.235,E2 -1542.235} C_VEL
LIN {X 0,Y 587.36,Z 294.902,A -85,B 0,C 180,E1 -1542.285,E2 -1542.285} C_VEL
LIN {X 0,Y 587.455,Z 275.124,A -85,B 0,C 180,E1 -1544.906,E2 -1544.906} C_VEL
LIN {X 0,Y 587.605,Z 255.18,A -85,B 0,C 180,E1 -1547.579,E2 -1547.579} C_VEL
LIN {X 0,Y 587.78,Z 233.906,A -85,B 0,C 180,E1 -1550.472,E2 -1550.472} C_VEL
LIN {X 0,Y 587.945,Z 213.962,A -85,B 0,C 180,E1 -1553.233,E2 -1553.233} C_VEL
LIN {X 0,Y 588.108,Z 193.938,A -85,B 0,C 180,E1 -1556.052,E2 -1556.052} C_VEL
LIN {X 0,Y 588.328,Z 175.585,A -85,B 0,C 180,E1 -1558.717,E2 -1558.717} C_VEL
LIN {X 0,Y 587.323,Z 170.33,A -85,B 0,C 180,E1 -1559.578,E2 -1559.578} C_VEL
LIN {X 0,Y 587.318,Z 170.327,A -85,B 0,C 180,E1 -1561.831,E2 -1561.831} C_VEL
LIN {X 0,Y 587.33,Z 170.323,A -85,B 0,C 180,E1 -1564.345,E2 -1564.345} C_VEL
LIN {X 0,Y 587.341,Z 170.32,A -85,B 0,C 180,E1 -1567.609,E2 -1567.609} C_VEL
LIN {X 0,Y 587.313,Z 170.331,A -85,B 0,C 180,E1 -1570.255,E2 -1570.255} C_VEL
LIN {X 0,Y 587.319,Z 170.323,A -85,B 0,C 180,E1 -1573.118,E2 -1573.118} C_VEL
LIN {X 0,Y 587.317,Z 170.325,A -85,B 0,C 180,E1 -1576.049,E2 -1576.049} C_VEL
LIN {X 0,Y 587.339,Z 170.325,A -85,B 0,C 180,E1 -1578.926,E2 -1578.926} C_VEL
LIN {X 0,Y 587.315,Z 170.324,A -85,B 0,C 180,E1 -1581.519,E2 -1581.519} C_VEL
LIN {X 0,Y 587.274,Z 170.332,A -85,B 0,C 180,E1 -1584.099,E2 -1584.099} C_VEL
LIN {X 0,Y 587.241,Z 170.529,A -85,B 0,C 180,E1 -1586.082,E2 -1586.082} C_VEL
LIN {X 0,Y 587.267,Z 179.951,A -85,B 0,C 180,E1 -1588.629,E2 -1588.629} C_VEL
LIN {X 0,Y 587.299,Z 189.493,A -85,B 0,C 180,E1 -1591.402,E2 -1591.402} C_VEL
LIN {X 0,Y 587.355,Z 198.298,A -85,B 0,C 180,E1 -1594.155,E2 -1594.155} C_VEL
LIN {X 0,Y 587.327,Z 206.2,A -85,B 0,C 180,E1 -1596.741,E2 -1596.741} C_VEL
LIN {X 0,Y 587.299,Z 214.005,A -85,B 0,C 180,E1 -1599.333,E2 -1599.333} C_VEL
LIN {X 0,Y 587.283,Z 222.891,A -85,B 0,C 180,E1 -1602.232,E2 -1602.232} C_VEL
LIN {X 0,Y 587.224,Z 231.794,A -85,B 0,C 180,E1 -1605.089,E2 -1605.089} C_VEL
LIN {X 0,Y 587.208,Z 240.488,A -85,B 0,C 180,E1 -1607.844,E2 -1607.844} C_VEL
LIN {X 0,Y 587.723,Z 246.363,A -85,B 0,C 180,E1 -1607.964,E2 -1607.964} C_VEL
LIN {X 0,Y 587.632,Z 259.948,A -85,B 0,C 180,E1 -1608.316,E2 -1608.316} C_VEL
LIN {X 0,Y 587.553,Z 272.534,A -85,B 0,C 180,E1 -1608.794,E2 -1608.794} C_VEL
LIN {X 0,Y 587.522,Z 284.529,A -85,B 0,C 180,E1 -1609.402,E2 -1609.402} C_VEL
LIN {X 0,Y 587.439,Z 295.326,A -85,B 0,C 180,E1 -1610.097,E2 -1610.097} C_VEL
LIN {X 0,Y 587.357,Z 305.101,A -85,B 0,C 180,E1 -1610.878,E2 -1610.878} C_VEL
LIN {X 0,Y 587.303,Z 313.997,A -85,B 0,C 180,E1 -1611.744,E2 -1611.744} C_VEL
LIN {X 0,Y 587.234,Z 322.666,A -85,B 0,C 180,E1 -1612.781,E2 -1612.781} C_VEL
LIN {X 0,Y 587.214,Z 329.61,A -85,B 0,C 180,E1 -1613.816,E2 -1613.816} C_VEL
LIN {X 0,Y 587.167,Z 335.164,A -85,B 0,C 180,E1 -1614.85,E2 -1614.85} C_VEL
LIN {X 0,Y 587.183,Z 339.523,A -85,B 0,C 180,E1 -1615.882,E2 -1615.882} C_VEL
LIN {X 0,Y 587.193,Z 341.824,A -85,B 0,C 180,E1 -1616.569,E2 -1616.569} C_VEL
LIN {X 0,Y 587.131,Z 343.692,A -85,B 0,C 180,E1 -1617.256,E2 -1617.256} C_VEL
LIN {X 0,Y 587.139,Z 345.131,A -85,B 0,C 180,E1 -1617.942,E2 -1617.942} C_VEL
LIN {X 0,Y 587.141,Z 346.754,A -85,B 0,C 180,E1 -1619.314,E2 -1619.314} C_VEL
LIN {X 0,Y 587.137,Z 346.996,A -85,B 0,C 180,E1 -1620,E2 -1620} C_VEL
LIN {X 0,Y 587.14,Z 346.814,A -85,B 0,C 180,E1 -1620.686,E2 -1620.686} C_VEL
LIN {X 0,Y 587.138,Z 345.275,A -85,B 0,C 180,E1 -1622.058,E2 -1622.058} C_VEL
LIN {X 0,Y 587.133,Z 343.913,A -85,B 0,C 180,E1 -1622.744,E2 -1622.744} C_VEL
LIN {X 0,Y 587.213,Z 341.042,A -85,B 0,C 180,E1 -1623.774,E2 -1623.774} C_VEL
LIN {X 0,Y 587.147,Z 337.144,A -85,B 0,C 180,E1 -1624.806,E2 -1624.806} C_VEL
LIN {X 0,Y 587.229,Z 332.108,A -85,B 0,C 180,E1 -1625.839,E2 -1625.839} C_VEL
LIN {X 0,Y 587.23,Z 325.775,A -85,B 0,C 180,E1 -1626.874,E2 -1626.874} C_VEL
LIN {X 0,Y 587.288,Z 317.872,A -85,B 0,C 180,E1 -1627.91,E2 -1627.91} C_VEL
LIN {X 0,Y 587.336,Z 309.801,A -85,B 0,C 180,E1 -1628.776,E2 -1628.776} C_VEL
LIN {X 0,Y 587.387,Z 299.954,A -85,B 0,C 180,E1 -1629.643,E2 -1629.643} C_VEL
LIN {X 0,Y 587.441,Z 288.898,A -85,B 0,C 180,E1 -1630.425,E2 -1630.425} C_VEL
LIN {X 0,Y 587.526,Z 277.035,A -85,B 0,C 180,E1 -1631.086,E2 -1631.086} C_VEL
LIN {X 0,Y 587.622,Z 265.324,A -85,B 0,C 180,E1 -1631.589,E2 -1631.589} C_VEL
LIN {X 0,Y 587.708,Z 252.259,A -85,B 0,C 180,E1 -1631.992,E2 -1631.992} C_VEL
LIN {X 0,Y 587.53,Z 242.988,A -85,B 0,C 180,E1 -1632.193,E2 -1632.193} C_VEL
LIN {X 0,Y 587.162,Z 240.495,A -85,B 0,C 180,E1 -1632.245,E2 -1632.245} C_VEL
LIN {X 0,Y 587.193,Z 238.073,A -85,B 0,C 180,E1 -1633.008,E2 -1633.008} C_VEL
LIN {X 0,Y 586.573,Z 236.385,A -85,B 0,C 180,E1 -1633.557,E2 -1633.557} C_VEL
LIN {X 0,Y 583.727,Z 233.795,A -85,B 0,C 180,E1 -1634.452,E2 -1634.452} C_VEL
LIN {X 0,Y 581.288,Z 231.749,A -85,B 0,C 180,E1 -1635.172,E2 -1635.172} C_VEL
LIN {X 0,Y 580.229,Z 230.122,A -85,B 0,C 180,E1 -1635.726,E2 -1635.726} C_VEL
LIN {X 0,Y 580.139,Z 229.551,A -85,B 0,C 180,E1 -1635.913,E2 -1635.913} C_VEL
LIN {X 0,Y 580.193,Z 220.941,A -85,B 0,C 180,E1 -1638.724,E2 -1638.724} C_VEL
LIN {X 0,Y 580.232,Z 212.034,A -85,B 0,C 180,E1 -1641.68,E2 -1641.68} C_VEL
LIN {X 0,Y 580.27,Z 204.206,A -85,B 0,C 180,E1 -1644.318,E2 -1644.318} C_VEL
LIN {X 0,Y 580.334,Z 196.352,A -85,B 0,C 180,E1 -1647.009,E2 -1647.009} C_VEL
LIN {X 0,Y 580.342,Z 187.938,A -85,B 0,C 180,E1 -1649.77,E2 -1649.77} C_VEL
LIN {X 0,Y 580.393,Z 180.603,A -85,B 0,C 180,E1 -1652.195,E2 -1652.195} C_VEL
LIN {X 0,Y 580.375,Z 171.866,A -85,B 0,C 180,E1 -1655.114,E2 -1655.114} C_VEL
LIN {X 0,Y 580.27,Z 171.206,A -85,B 0,C 180,E1 -1655.44,E2 -1655.44} C_VEL
LIN {X 0,Y 580.286,Z 171.203,A -85,B 0,C 180,E1 -1658.147,E2 -1658.147} C_VEL
LIN {X 0,Y 580.301,Z 171.202,A -85,B 0,C 180,E1 -1660.843,E2 -1660.843} C_VEL
LIN {X 0,Y 580.245,Z 171.205,A -85,B 0,C 180,E1 -1663.661,E2 -1663.661} C_VEL
LIN {X 0,Y 580.278,Z 171.201,A -85,B 0,C 180,E1 -1666.61,E2 -1666.61} C_VEL
LIN {X 0,Y 580.302,Z 171.205,A -85,B 0,C 180,E1 -1669.156,E2 -1669.156} C_VEL
LIN {X 0,Y 580.285,Z 171.202,A -85,B 0,C 180,E1 -1671.928,E2 -1671.928} C_VEL
LIN {X 0,Y 580.23,Z 171.208,A -85,B 0,C 180,E1 -1674.45,E2 -1674.45} C_VEL
LIN {X 0,Y 580.293,Z 171.204,A -85,B 0,C 180,E1 -1676.975,E2 -1676.975} C_VEL
LIN {X 0,Y 580.301,Z 171.199,A -85,B 0,C 180,E1 -1679.425,E2 -1679.425} C_VEL
LIN {X 0,Y 580.196,Z 171.326,A -85,B 0,C 180,E1 -1680.71,E2 -1680.71} C_VEL
LIN {X 0,Y 580.193,Z 174.924,A -85,B 0,C 180,E1 -1683.372,E2 -1683.372} C_VEL
LIN {X 0,Y 580.143,Z 178.03,A -85,B 0,C 180,E1 -1685.676,E2 -1685.676} C_VEL
LIN {X 0,Y 580.116,Z 181.096,A -85,B 0,C 180,E1 -1687.94,E2 -1687.94} C_VEL
LIN {X 0,Y 580.06,Z 184.131,A -85,B 0,C 180,E1 -1690.168,E2 -1690.168} C_VEL
LIN {X 0,Y 580.041,Z 187.17,A -85,B 0,C 180,E1 -1692.367,E2 -1692.367} C_VEL
LIN {X 0,Y 580.047,Z 190.475,A -85,B 0,C 180,E1 -1694.54,E2 -1694.54} C_VEL
LIN {X 0,Y 580.048,Z 193.779,A -85,B 0,C 180,E1 -1696.69,E2 -1696.69} C_VEL
LIN {X 0,Y 580.043,Z 198.185,A -85,B 0,C 180,E1 -1699.528,E2 -1699.528} C_VEL
LIN {X 0,Y 580.019,Z 203.141,A -85,B 0,C 180,E1 -1702.69,E2 -1702.69} C_VEL
LIN {X 0,Y 580.044,Z 203.451,A -85,B 0,C 180,E1 -1702.887,E2 -1702.887} C_VEL
LIN {X 0,Y 580.239,Z 211.46,A -85,B 0,C 180,E1 -1703.191,E2 -1703.191} C_VEL
LIN {X 0,Y 580.22,Z 219.249,A -85,B 0,C 180,E1 -1703.582,E2 -1703.582} C_VEL
LIN {X 0,Y 580.145,Z 226.976,A -85,B 0,C 180,E1 -1704.089,E2 -1704.089} C_VEL
LIN {X 0,Y 580.118,Z 233.233,A -85,B 0,C 180,E1 -1704.612,E2 -1704.612} C_VEL
LIN {X 0,Y 580.182,Z 239.789,A -85,B 0,C 180,E1 -1705.309,E2 -1705.309} C_VEL
LIN {X 0,Y 580.133,Z 244.911,A -85,B 0,C 180,E1 -1706.005,E2 -1706.005} C_VEL
LIN {X 0,Y 580.095,Z 249.816,A -85,B 0,C 180,E1 -1706.874,E2 -1706.874} C_VEL
LIN {X 0,Y 580.048,Z 253.849,A -85,B 0,C 180,E1 -1707.916,E2 -1707.916} C_VEL
LIN {X 0,Y 580.047,Z 255.566,A -85,B 0,C 180,E1 -1708.611,E2 -1708.611} C_VEL
LIN {X 0,Y 580.041,Z 256.584,A -85,B 0,C 180,E1 -1709.305,E2 -1709.305} C_VEL
LIN {X 0,Y 580.038,Z 256.957,A -85,B 0,C 180,E1 -1709.999,E2 -1709.999} C_VEL
LIN {X 0,Y 580.04,Z 256.693,A -85,B 0,C 180,E1 -1710.693,E2 -1710.693} C_VEL
LIN {X 0,Y 580.048,Z 255.764,A -85,B 0,C 180,E1 -1711.388,E2 -1711.388} C_VEL
LIN {X 0,Y 580.092,Z 253.005,A -85,B 0,C 180,E1 -1712.429,E2 -1712.429} C_VEL
LIN {X 0,Y 580.095,Z 250.252,A -85,B 0,C 180,E1 -1713.124,E2 -1713.124} C_VEL
LIN {X 0,Y 580.133,Z 245.518,A -85,B 0,C 180,E1 -1713.993,E2 -1713.993} C_VEL
LIN {X 0,Y 580.169,Z 240.548,A -85,B 0,C 180,E1 -1714.689,E2 -1714.689} C_VEL
LIN {X 0,Y 580.112,Z 234.207,A -85,B 0,C 180,E1 -1715.387,E2 -1715.387} C_VEL
LIN {X 0,Y 580.149,Z 227.038,A -85,B 0,C 180,E1 -1715.997,E2 -1715.997} C_VEL
LIN {X 0,Y 580.167,Z 220.303,A -85,B 0,C 180,E1 -1716.448,E2 -1716.448} C_VEL
LIN {X 0,Y 580.275,Z 211.779,A -85,B 0,C 180,E1 -1716.885,E2 -1716.885} C_VEL
LIN {X 0,Y 580.092,Z 204.019,A -85,B 0,C 180,E1 -1717.176,E2 -1717.176} C_VEL
LIN {X 0,Y 580.033,Z 203.423,A -85,B 0,C 180,E1 -1717.221,E2 -1717.221} C_VEL
LIN {X 0,Y 580.037,Z 198.328,A -85,B 0,C 180,E1 -1720.471,E2 -1720.471} C_VEL
LIN {X 0,Y 580.04,Z 193.921,A -85,B 0,C 180,E1 -1723.308,E2 -1723.308} C_VEL
LIN {X 0,Y 580.072,Z 189.513,A -85,B 0,C 180,E1 -1726.179,E2 -1726.179} C_VEL
LIN {X 0,Y 580.057,Z 185.227,A -85,B 0,C 180,E1 -1729.094,E2 -1729.094} C_VEL
LIN {X 0,Y 580.087,Z 182.242,A -85,B 0,C 180,E1 -1731.312,E2 -1731.312} C_VEL
LIN {X 0,Y 580.131,Z 179.195,A -85,B 0,C 180,E1 -1733.563,E2 -1733.563} C_VEL
LIN {X 0,Y 580.207,Z 175.477,A -85,B 0,C 180,E1 -1736.316,E2 -1736.316} C_VEL
LIN {X 0,Y 580.222,Z 171.869,A -85,B 0,C 180,E1 -1738.979,E2 -1738.979} C_VEL
LIN {X 0,Y 580.237,Z 171.212,A -85,B 0,C 180,E1 -1739.774,E2 -1739.774} C_VEL
LIN {X 0,Y 580.292,Z 171.198,A -85,B 0,C 180,E1 -1742.2,E2 -1742.2} C_VEL
LIN {X 0,Y 580.284,Z 171.198,A -85,B 0,C 180,E1 -1744.695,E2 -1744.695} C_VEL
LIN {X 0,Y 580.293,Z 171.204,A -85,B 0,C 180,E1 -1747.267,E2 -1747.267} C_VEL
LIN {X 0,Y 580.29,Z 171.197,A -85,B 0,C 180,E1 -1750.27,E2 -1750.27} C_VEL
LIN {X 0,Y 580.275,Z 171.202,A -85,B 0,C 180,E1 -1752.705,E2 -1752.705} C_VEL
LIN {X 0,Y 580.263,Z 171.201,A -85,B 0,C 180,E1 -1755.608,E2 -1755.608} C_VEL
LIN {X 0,Y 580.307,Z 171.196,A -85,B 0,C 180,E1 -1758.233,E2 -1758.233} C_VEL
LIN {X 0,Y 580.283,Z 171.204,A -85,B 0,C 180,E1 -1760.965,E2 -1760.965} C_VEL
LIN {X 0,Y 580.289,Z 171.196,A -85,B 0,C 180,E1 -1763.598,E2 -1763.598} C_VEL
LIN {X 0,Y 580.314,Z 171.197,A -85,B 0,C 180,E1 -1766.145,E2 -1766.145} C_VEL
LIN {X 0,Y 580.283,Z 171.203,A -85,B 0,C 180,E1 -1768.615,E2 -1768.615} C_VEL
LIN {X 0,Y 580.289,Z 171.197,A -85,B 0,C 180,E1 -1771.024,E2 -1771.024} C_VEL
LIN {X 0,Y 580.319,Z 171.195,A -85,B 0,C 180,E1 -1773.658,E2 -1773.658} C_VEL
LIN {X 0,Y 580.273,Z 171.202,A -85,B 0,C 180,E1 -1776.442,E2 -1776.442} C_VEL
LIN {X 0,Y 580.274,Z 171.201,A -85,B 0,C 180,E1 -1779.437,E2 -1779.437} C_VEL
LIN {X 0,Y 580.272,Z 171.205,A -85,B 0,C 180,E1 -1781.645,E2 -1781.645} C_VEL
LIN {X 0,Y 580.274,Z 171.205,A -85,B 0,C 180,E1 -1783.825,E2 -1783.825} C_VEL
LIN {X 0,Y 580.271,Z 171.199,A -85,B 0,C 180,E1 -1786.696,E2 -1786.696} C_VEL
LIN {X 0,Y 580.293,Z 171.203,A -85,B 0,C 180,E1 -1789.533,E2 -1789.533} C_VEL
LIN {X 0,Y 580.322,Z 171.192,A -85,B 0,C 180,E1 -1792.344,E2 -1792.344} C_VEL
LIN {X 0,Y 580.327,Z 171.2,A -85,B 0,C 180,E1 -1795.137,E2 -1795.137} C_VEL
LIN {X 0,Y 580.315,Z 171.193,A -85,B 0,C 180,E1 -1797.918,E2 -1797.918} C_VEL
LIN {X 0,Y 580.361,Z 171.192,A -85,B 0,C 180,E1 -1800.694,E2 -1800.694} C_VEL
LIN {X 0,Y 580.257,Z 171.201,A -85,B 0,C 180,E1 -1803.472,E2 -1803.472} C_VEL
LIN {X 0,Y 580.296,Z 171.195,A -85,B 0,C 180,E1 -1805.56,E2 -1805.56} C_VEL
LIN {X 0,Y 580.318,Z 171.199,A -85,B 0,C 180,E1 -1808.356,E2 -1808.356} C_VEL
LIN {X 0,Y 580.288,Z 171.197,A -85,B 0,C 180,E1 -1811.191,E2 -1811.191} C_VEL
LIN {X 0,Y 580.308,Z 171.198,A -85,B 0,C 180,E1 -1814.017,E2 -1814.017} C_VEL
LIN {X 0,Y 580.277,Z 171.198,A -85,B 0,C 180,E1 -1816.907,E2 -1816.907} C_VEL
LIN {X 0,Y 580.264,Z 171.206,A -85,B 0,C 180,E1 -1819.824,E2 -1819.824} C_VEL
LIN {X 0,Y 580.236,Z 171.212,A -85,B 0,C 180,E1 -1822.054,E2 -1822.054} C_VEL
LIN {X 0,Y 580.263,Z 171.201,A -85,B 0,C 180,E1 -1825.082,E2 -1825.082} C_VEL
LIN {X 0,Y 580.227,Z 171.212,A -85,B 0,C 180,E1 -1827.848,E2 -1827.848} C_VEL
LIN {X 0,Y 580.254,Z 171.201,A -85,B 0,C 180,E1 -1830.692,E2 -1830.692} C_VEL
LIN {X 0,Y 580.289,Z 171.204,A -85,B 0,C 180,E1 -1833.317,E2 -1833.317} C_VEL
LIN {X 0,Y 580.219,Z 171.209,A -85,B 0,C 180,E1 -1835.755,E2 -1835.755} C_VEL
LIN {X 0,Y 580.271,Z 171.2,A -85,B 0,C 180,E1 -1838.148,E2 -1838.148} C_VEL
LIN {X 0,Y 580.287,Z 171.202,A -85,B 0,C 180,E1 -1840.845,E2 -1840.845} C_VEL
LIN {X 0,Y 580.262,Z 171.201,A -85,B 0,C 180,E1 -1843.66,E2 -1843.66} C_VEL
LIN {X 0,Y 580.266,Z 171.206,A -85,B 0,C 180,E1 -1846.611,E2 -1846.611} C_VEL
LIN {X 0,Y 580.291,Z 171.2,A -85,B 0,C 180,E1 -1849.158,E2 -1849.158} C_VEL
LIN {X 0,Y 580.28,Z 171.2,A -85,B 0,C 180,E1 -1851.929,E2 -1851.929} C_VEL
LIN {X 0,Y 580.25,Z 171.211,A -85,B 0,C 180,E1 -1854.454,E2 -1854.454} C_VEL
LIN {X 0,Y 580.285,Z 171.201,A -85,B 0,C 180,E1 -1856.976,E2 -1856.976} C_VEL
LIN {X 0,Y 580.272,Z 171.206,A -85,B 0,C 180,E1 -1859.827,E2 -1859.827} C_VEL
LIN {X 0,Y 580.308,Z 171.27,A -85,B 0,C 180,E1 -1860.18,E2 -1860.18} C_VEL
LIN {X 0,Y 581.46,Z 176.709,A -85,B 0,C 180,E1 -1861.089,E2 -1861.089} C_VEL
LIN {X 0,Y 581.275,Z 192.825,A -85,B 0,C 180,E1 -1863.471,E2 -1863.471} C_VEL
LIN {X 0,Y 581.109,Z 211.31,A -85,B 0,C 180,E1 -1866.101,E2 -1866.101} C_VEL
LIN {X 0,Y 580.866,Z 231.261,A -85,B 0,C 180,E1 -1868.904,E2 -1868.904} C_VEL
LIN {X 0,Y 580.688,Z 252.534,A -85,B 0,C 180,E1 -1871.842,E2 -1871.842} C_VEL
LIN {X 0,Y 580.492,Z 272.478,A -85,B 0,C 180,E1 -1874.554,E2 -1874.554} C_VEL
LIN {X 0,Y 580.387,Z 292.422,A -85,B 0,C 180,E1 -1877.234,E2 -1877.234} C_VEL
LIN {X 0,Y 580.342,Z 294.915,A -85,B 0,C 180,E1 -1877.566,E2 -1877.566} C_VEL
LIN {X 0,Y 580.82,Z 300.174,A -85,B 0,C 180,E1 -1877.665,E2 -1877.665} C_VEL
LIN {X 0,Y 580.742,Z 313.132,A -85,B 0,C 180,E1 -1877.929,E2 -1877.929} C_VEL
LIN {X 0,Y 580.646,Z 325.438,A -85,B 0,C 180,E1 -1878.321,E2 -1878.321} C_VEL
LIN {X 0,Y 580.592,Z 337.199,A -85,B 0,C 180,E1 -1878.833,E2 -1878.833} C_VEL
LIN {X 0,Y 580.476,Z 349.602,A -85,B 0,C 180,E1 -1879.537,E2 -1879.537} C_VEL
LIN {X 0,Y 580.379,Z 360.485,A -85,B 0,C 180,E1 -1880.328,E2 -1880.328} C_VEL
LIN {X 0,Y 580.271,Z 371.123,A -85,B 0,C 180,E1 -1881.293,E2 -1881.293} C_VEL
LIN {X 0,Y 580.221,Z 378.968,A -85,B 0,C 180,E1 -1882.169,E2 -1882.169} C_VEL
LIN {X 0,Y 580.153,Z 386.656,A -85,B 0,C 180,E1 -1883.222,E2 -1883.222} C_VEL
LIN {X 0,Y 580.139,Z 393.685,A -85,B 0,C 180,E1 -1884.439,E2 -1884.439} C_VEL
LIN {X 0,Y 580.108,Z 398.375,A -85,B 0,C 180,E1 -1885.484,E2 -1885.484} C_VEL
LIN {X 0,Y 580.122,Z 401.961,A -85,B 0,C 180,E1 -1886.528,E2 -1886.528} C_VEL
LIN {X 0,Y 580.043,Z 403.812,A -85,B 0,C 180,E1 -1887.223,E2 -1887.223} C_VEL
LIN {X 0,Y 580.04,Z 405.202,A -85,B 0,C 180,E1 -1887.918,E2 -1887.918} C_VEL
LIN {X 0,Y 580.04,Z 406.785,A -85,B 0,C 180,E1 -1889.307,E2 -1889.307} C_VEL
LIN {X 0,Y 580.037,Z 407,A -85,B 0,C 180,E1 -1890.001,E2 -1890.001} C_VEL
LIN {X 0,Y 580.047,Z 406.184,A -85,B 0,C 180,E1 -1891.389,E2 -1891.389} C_VEL
LIN {X 0,Y 580.04,Z 405.198,A -85,B 0,C 180,E1 -1892.084,E2 -1892.084} C_VEL
LIN {X 0,Y 580.043,Z 403.806,A -85,B 0,C 180,E1 -1892.779,E2 -1892.779} C_VEL
LIN {X 0,Y 580.11,Z 400.893,A -85,B 0,C 180,E1 -1893.821,E2 -1893.821} C_VEL
LIN {X 0,Y 580.053,Z 396.946,A -85,B 0,C 180,E1 -1894.866,E2 -1894.866} C_VEL
LIN {X 0,Y 580.139,Z 390.872,A -85,B 0,C 180,E1 -1896.086,E2 -1896.086} C_VEL
LIN {X 0,Y 580.185,Z 384.231,A -85,B 0,C 180,E1 -1897.133,E2 -1897.133} C_VEL
LIN {X 0,Y 580.251,Z 375.983,A -85,B 0,C 180,E1 -1898.183,E2 -1898.183} C_VEL
LIN {X 0,Y 580.308,Z 367.529,A -85,B 0,C 180,E1 -1899.059,E2 -1899.059} C_VEL
LIN {X 0,Y 580.42,Z 357.087,A -85,B 0,C 180,E1 -1899.937,E2 -1899.937} C_VEL
LIN {X 0,Y 580.5,Z 346.742,A -85,B 0,C 180,E1 -1900.64,E2 -1900.64} C_VEL
LIN {X 0,Y 580.582,Z 335.399,A -85,B 0,C 180,E1 -1901.257,E2 -1901.257} C_VEL
LIN {X 0,Y 580.668,Z 323.749,A -85,B 0,C 180,E1 -1901.742,E2 -1901.742} C_VEL
LIN {X 0,Y 580.768,Z 310.32,A -85,B 0,C 180,E1 -1902.138,E2 -1902.138} C_VEL
LIN {X 0,Y 580.668,Z 297.227,A -85,B 0,C 180,E1 -1902.382,E2 -1902.382} C_VEL
LIN {X 0,Y 580.343,Z 294.902,A -85,B 0,C 180,E1 -1902.436,E2 -1902.436} C_VEL
LIN {X 0,Y 580.458,Z 275.124,A -85,B 0,C 180,E1 -1905.09,E2 -1905.09} C_VEL
LIN {X 0,Y 580.639,Z 255.18,A -85,B 0,C 180,E1 -1907.796,E2 -1907.796} C_VEL
LIN {X 0,Y 580.84,Z 235.236,A -85,B 0,C 180,E1 -1910.543,E2 -1910.543} C_VEL
LIN {X 0,Y 581.055,Z 215.615,A -85,B 0,C 180,E1 -1913.291,E2 -1913.291} C_VEL
LIN {X 0,Y 581.23,Z 195.197,A -85,B 0,C 180,E1 -1916.176,E2 -1916.176} C_VEL
LIN {X 0,Y 581.524,Z 177.991,A -85,B 0,C 180,E1 -1918.712,E2 -1918.712} C_VEL
LIN {X 0,Y 580.29,Z 171.206,A -85,B 0,C 180,E1 -1919.836,E2 -1919.836} C_VEL
LIN {X 0,Y 580.281,Z 171.202,A -85,B 0,C 180,E1 -1922.202,E2 -1922.202} C_VEL
LIN {X 0,Y 580.277,Z 171.206,A -85,B 0,C 180,E1 -1924.698,E2 -1924.698} C_VEL
LIN {X 0,Y 580.289,Z 171.2,A -85,B 0,C 180,E1 -1927.27,E2 -1927.27} C_VEL
LIN {X 0,Y 580.292,Z 171.206,A -85,B 0,C 180,E1 -1930.27,E2 -1930.27} C_VEL
LIN {X 0,Y 580.282,Z 171.2,A -85,B 0,C 180,E1 -1932.707,E2 -1932.707} C_VEL
LIN {X 0,Y 580.26,Z 171.21,A -85,B 0,C 180,E1 -1935.611,E2 -1935.611} C_VEL
LIN {X 0,Y 580.281,Z 171.2,A -85,B 0,C 180,E1 -1938.231,E2 -1938.231} C_VEL
LIN {X 0,Y 580.27,Z 171.209,A -85,B 0,C 180,E1 -1940.964,E2 -1940.964} C_VEL
LIN {X 0,Y 580.243,Z 171.205,A -85,B 0,C 180,E1 -1943.594,E2 -1943.594} C_VEL
LIN {X 0,Y 580.202,Z 171.3,A -85,B 0,C 180,E1 -1946.085,E2 -1946.085} C_VEL
LIN {X 0,Y 580.218,Z 180.617,A -85,B 0,C 180,E1 -1948.611,E2 -1948.611} C_VEL
LIN {X 0,Y 580.252,Z 190.267,A -85,B 0,C 180,E1 -1951.417,E2 -1951.417} C_VEL
LIN {X 0,Y 580.296,Z 199.092,A -85,B 0,C 180,E1 -1954.151,E2 -1954.151} C_VEL
LIN {X 0,Y 580.298,Z 206.105,A -85,B 0,C 180,E1 -1956.443,E2 -1956.443} C_VEL
LIN {X 0,Y 580.243,Z 215.104,A -85,B 0,C 180,E1 -1959.436,E2 -1959.436} C_VEL
LIN {X 0,Y 580.207,Z 224.006,A -85,B 0,C 180,E1 -1962.373,E2 -1962.373} C_VEL
LIN {X 0,Y 580.156,Z 232.908,A -85,B 0,C 180,E1 -1965.262,E2 -1965.262} C_VEL
LIN {X 0,Y 580.161,Z 240.717,A -85,B 0,C 180,E1 -1967.705,E2 -1967.705} C_VEL
LIN {X 0,Y 580.787,Z 246.407,A -85,B 0,C 180,E1 -1967.819,E2 -1967.819} C_VEL
LIN {X 0,Y 580.703,Z 259.863,A -85,B 0,C 180,E1 -1968.171,E2 -1968.171} C_VEL
LIN {X 0,Y 580.579,Z 272.894,A -85,B 0,C 180,E1 -1968.673,E2 -1968.673} C_VEL
LIN {X 0,Y 580.535,Z 284.538,A -85,B 0,C 180,E1 -1969.273,E2 -1969.273} C_VEL
LIN {X 0,Y 580.447,Z 295.332,A -85,B 0,C 180,E1 -1969.977,E2 -1969.977} C_VEL
LIN {X 0,Y 580.333,Z 305.106,A -85,B 0,C 180,E1 -1970.766,E2 -1970.766} C_VEL
LIN {X 0,Y 580.265,Z 314.004,A -85,B 0,C 180,E1 -1971.643,E2 -1971.643} C_VEL
LIN {X 0,Y 580.176,Z 322.667,A -85,B 0,C 180,E1 -1972.693,E2 -1972.693} C_VEL
LIN {X 0,Y 580.137,Z 329.615,A -85,B 0,C 180,E1 -1973.741,E2 -1973.741} C_VEL
LIN {X 0,Y 580.086,Z 335.169,A -85,B 0,C 180,E1 -1974.787,E2 -1974.787} C_VEL
LIN {X 0,Y 580.106,Z 339.527,A -85,B 0,C 180,E1 -1975.832,E2 -1975.832} C_VEL
LIN {X 0,Y 580.123,Z 341.828,A -85,B 0,C 180,E1 -1976.527,E2 -1976.527} C_VEL
LIN {X 0,Y 580.043,Z 343.691,A -85,B 0,C 180,E1 -1977.222,E2 -1977.222} C_VEL
LIN {X 0,Y 580.038,Z 345.132,A -85,B 0,C 180,E1 -1977.917,E2 -1977.917} C_VEL
LIN {X 0,Y 580.041,Z 346.754,A -85,B 0,C 180,E1 -1979.306,E2 -1979.306} C_VEL
LIN {X 0,Y 580.038,Z 346.996,A -85,B 0,C 180,E1 -1980,E2 -1980} C_VEL
LIN {X 0,Y 580.04,Z 346.814,A -85,B 0,C 180,E1 -1980.694,E2 -1980.694} C_VEL
LIN {X 0,Y 580.037,Z 345.275,A -85,B 0,C 180,E1 -1982.083,E2 -1982.083} C_VEL
LIN {X 0,Y 580.044,Z 343.911,A -85,B 0,C 180,E1 -1982.778,E2 -1982.778} C_VEL
LIN {X 0,Y 580.11,Z 341.041,A -85,B 0,C 180,E1 -1983.821,E2 -1983.821} C_VEL
LIN {X 0,Y 580.054,Z 337.143,A -85,B 0,C 180,E1 -1984.865,E2 -1984.865} C_VEL
LIN {X 0,Y 580.162,Z 332.103,A -85,B 0,C 180,E1 -1985.91,E2 -1985.91} C_VEL
LIN {X 0,Y 580.158,Z 325.769,A -85,B 0,C 180,E1 -1986.958,E2 -1986.958} C_VEL
LIN {X 0,Y 580.242,Z 317.87,A -85,B 0,C 180,E1 -1988.007,E2 -1988.007} C_VEL
LIN {X 0,Y 580.305,Z 309.797,A -85,B 0,C 180,E1 -1988.883,E2 -1988.883} C_VEL
LIN {X 0,Y 580.365,Z 299.945,A -85,B 0,C 180,E1 -1989.761,E2 -1989.761} C_VEL
LIN {X 0,Y 580.453,Z 288.89,A -85,B 0,C 180,E1 -1990.552,E2 -1990.552} C_VEL
LIN {X 0,Y 580.551,Z 278.069,A -85,B 0,C 180,E1 -1991.168,E2 -1991.168} C_VEL
LIN {X 0,Y 580.652,Z 266.154,A -85,B 0,C 180,E1 -1991.697,E2 -1991.697} C_VEL
LIN {X 0,Y 580.751,Z 253.077,A -85,B 0,C 180,E1 -1992.116,E2 -1992.116} C_VEL
LIN {X 0,Y 580.56,Z 243.436,A -85,B 0,C 180,E1 -1992.333,E2 -1992.333} C_VEL
LIN {X 0,Y 580.107,Z 240.493,A -85,B 0,C 180,E1 -1992.396,E2 -1992.396} C_VEL
LIN {X 0,Y 580.146,Z 232.074,A -85,B 0,C 180,E1 -1995.097,E2 -1995.097} C_VEL
LIN {X 0,Y 580.139,Z 229.551,A -85,B 0,C 180,E1 -1995.913,E2 -1995.913} C_VEL
LIN {X 0,Y 579.46,Z 227.898,A -85,B 0,C 180,E1 -1996.47,E2 -1996.47} C_VEL
LIN {X 0,Y 576.605,Z 225.383,A -85,B 0,C 180,E1 -1997.378,E2 -1997.378} C_VEL
LIN {X 0,Y 574.217,Z 223.396,A -85,B 0,C 180,E1 -1998.11,E2 -1998.11} C_VEL
LIN {X 0,Y 573.214,Z 221.803,A -85,B 0,C 180,E1 -1998.672,E2 -1998.672} C_VEL
LIN {X 0,Y 573.143,Z 221.241,A -85,B 0,C 180,E1 -1998.862,E2 -1998.862} C_VEL
LIN {X 0,Y 573.202,Z 213.207,A -85,B 0,C 180,E1 -2001.582,E2 -2001.582} C_VEL
LIN {X 0,Y 573.239,Z 205.289,A -85,B 0,C 180,E1 -2004.25,E2 -2004.25} C_VEL
LIN {X 0,Y 573.307,Z 197.344,A -85,B 0,C 180,E1 -2006.973,E2 -2006.973} C_VEL
LIN {X 0,Y 573.296,Z 189.741,A -85,B 0,C 180,E1 -2009.496,E2 -2009.496} C_VEL
LIN {X 0,Y 573.333,Z 182.794,A -85,B 0,C 180,E1 -2011.81,E2 -2011.81} C_VEL
LIN {X 0,Y 573.384,Z 173.952,A -85,B 0,C 180,E1 -2014.792,E2 -2014.792} C_VEL
LIN {X 0,Y 573.219,Z 172.085,A -85,B 0,C 180,E1 -2015.456,E2 -2015.456} C_VEL
LIN {X 0,Y 573.229,Z 172.081,A -85,B 0,C 180,E1 -2018.31,E2 -2018.31} C_VEL
LIN {X 0,Y 573.25,Z 172.077,A -85,B 0,C 180,E1 -2020.525,E2 -2020.525} C_VEL
LIN {X 0,Y 573.212,Z 172.081,A -85,B 0,C 180,E1 -2023.362,E2 -2023.362} C_VEL
LIN {X 0,Y 573.243,Z 172.079,A -85,B 0,C 180,E1 -2026.332,E2 -2026.332} C_VEL
LIN {X 0,Y 573.234,Z 172.079,A -85,B 0,C 180,E1 -2028.543,E2 -2028.543} C_VEL
LIN {X 0,Y 573.241,Z 172.078,A -85,B 0,C 180,E1 -2031.298,E2 -2031.298} C_VEL
LIN {X 0,Y 573.189,Z 172.09,A -85,B 0,C 180,E1 -2034.022,E2 -2034.022} C_VEL
LIN {X 0,Y 573.236,Z 172.079,A -85,B 0,C 180,E1 -2036.515,E2 -2036.515} C_VEL
LIN {X 0,Y 573.234,Z 172.081,A -85,B 0,C 180,E1 -2039.118,E2 -2039.118} C_VEL
LIN {X 0,Y 573.154,Z 172.095,A -85,B 0,C 180,E1 -2040.627,E2 -2040.627} C_VEL
LIN {X 0,Y 573.143,Z 175.21,A -85,B 0,C 180,E1 -2043.018,E2 -2043.018} C_VEL
LIN {X 0,Y 573.124,Z 178.336,A -85,B 0,C 180,E1 -2045.358,E2 -2045.358} C_VEL
LIN {X 0,Y 573.048,Z 181.42,A -85,B 0,C 180,E1 -2047.654,E2 -2047.654} C_VEL
LIN {X 0,Y 573.003,Z 184.499,A -85,B 0,C 180,E1 -2049.914,E2 -2049.914} C_VEL
LIN {X 0,Y 572.977,Z 188.442,A -85,B 0,C 180,E1 -2052.879,E2 -2052.879} C_VEL
LIN {X 0,Y 572.986,Z 192.678,A -85,B 0,C 180,E1 -2055.799,E2 -2055.799} C_VEL
LIN {X 0,Y 572.984,Z 197.402,A -85,B 0,C 180,E1 -2058.888,E2 -2058.888} C_VEL
LIN {X 0,Y 572.916,Z 201.49,A -85,B 0,C 180,E1 -2061.534,E2 -2061.534} C_VEL
LIN {X 0,Y 572.941,Z 203.452,A -85,B 0,C 180,E1 -2062.798,E2 -2062.798} C_VEL
LIN {X 0,Y 573.23,Z 209.93,A -85,B 0,C 180,E1 -2063.04,E2 -2063.04} C_VEL
LIN {X 0,Y 573.165,Z 218.189,A -85,B 0,C 180,E1 -2063.441,E2 -2063.441} C_VEL
LIN {X 0,Y 573.115,Z 225.799,A -85,B 0,C 180,E1 -2063.928,E2 -2063.928} C_VEL
LIN {X 0,Y 573.032,Z 233.224,A -85,B 0,C 180,E1 -2064.545,E2 -2064.545} C_VEL
LIN {X 0,Y 573.091,Z 238.318,A -85,B 0,C 180,E1 -2065.075,E2 -2065.075} C_VEL
LIN {X 0,Y 573.037,Z 243.754,A -85,B 0,C 180,E1 -2065.779,E2 -2065.779} C_VEL
LIN {X 0,Y 573.062,Z 248.047,A -85,B 0,C 180,E1 -2066.484,E2 -2066.484} C_VEL
LIN {X 0,Y 572.973,Z 251.373,A -85,B 0,C 180,E1 -2067.187,E2 -2067.187} C_VEL
LIN {X 0,Y 572.951,Z 253.854,A -85,B 0,C 180,E1 -2067.89,E2 -2067.89} C_VEL
LIN {X 0,Y 572.947,Z 255.566,A -85,B 0,C 180,E1 -2068.593,E2 -2068.593} C_VEL
LIN {X 0,Y 572.941,Z 256.577,A -85,B 0,C 180,E1 -2069.296,E2 -2069.296} C_VEL
LIN {X 0,Y 572.938,Z 256.947,A -85,B 0,C 180,E1 -2069.999,E2 -2069.999} C_VEL
LIN {X 0,Y 572.941,Z 256.684,A -85,B 0,C 180,E1 -2070.702,E2 -2070.702} C_VEL
LIN {X 0,Y 572.948,Z 255.763,A -85,B 0,C 180,E1 -2071.405,E2 -2071.405} C_VEL
